KUKA KRL program: MyProgram_222().src

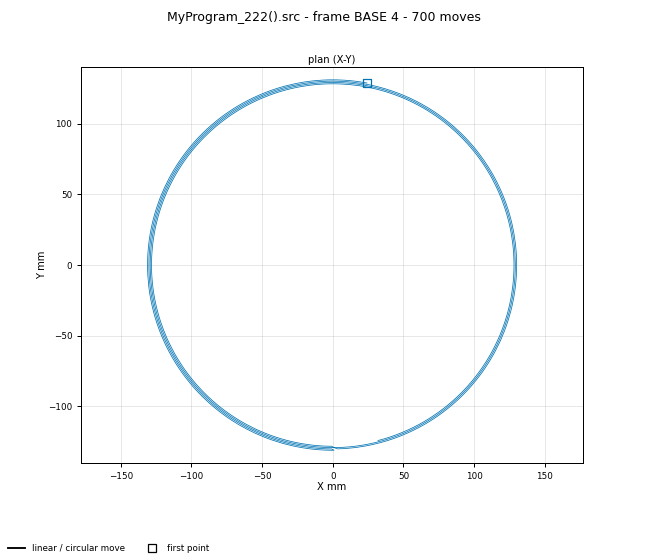
[picture p0: tool path of MyProgram_222().src in frame BASE 4, 700 of 700 moves have a stored position in this frame; points joined in program order, loops and branches not executed]
&ACCESS RVP
&REL 1
&PARAM TEMPLATE = C:\KRC\Roboter\Template\vorgabe
&PARAM EDITMASK = *
DEF MyProgram_222()
; ---- Setting reference (Base) ----
$BASE = BASE_DATA[4]

; --------------------------
; ---- Setting tool (TCP) ----
$TOOL = TOOL_DATA[3]
; --------------------------

$VEL.CP = VEL_APROX_PRINT
Startdeposition()
$VEL.CP = VEL_PRINT
LIN {X 24.2345,Y 128.7731,Z 154,A 76.9385,B 20.8095,C -0.9672,E1 20.8599,E2 370.7346} C_DIS
LIN {X 21.4392,Y 129.2675,Z 154,A 78.2158,B 20.8094,C -0.9692,E1 20.8564,E2 369.4533} C_DIS
LIN {X 16.024,Y 130.0508,Z 154,A 80.7871,B 20.809,C -0.9774,E1 20.8492,E2 366.8615} C_DIS
LIN {X 11.868,Y 130.4964,Z 154,A 82.5489,B 20.8091,C -0.9749,E1 20.8444,E2 365.1082} C_DIS
LIN {X 8.0216,Y 130.7876,Z 154,A 84.1635,B 20.8092,C -0.972,E1 20.8399,E2 363.5027} C_DIS
LIN {X 2.5644,Y 131.0089,Z 154,A 86.3389,B 20.8096,C -0.9629,E1 20.8339,E2 361.3536} C_DIS
LIN {X -2.8562,Y 131.0038,Z 154,A 88.8377,B 20.8094,C -0.9678,E1 20.8269,E2 358.8408} C_DIS
LIN {X -6.3957,Y 130.8773,Z 154,A 90.456,B 20.8094,C -0.9703,E1 20.8224,E2 357.2152} C_DIS
LIN {X -11.494,Y 130.529,Z 154,A 92.9422,B 20.8089,C -0.98,E1 20.8154,E2 354.7005} C_DIS
LIN {X -16.5105,Y 129.9899,Z 154,A 94.7586,B 20.8097,C -0.9625,E1 20.8104,E2 352.9318} C_DIS
LIN {X -20.6648,Y 129.3949,Z 154,A 97.517,B 20.808,C -0.9999,E1 20.8026,E2 350.065} C_DIS
LIN {X -26.2487,Y 128.3772,Z 154,A 99.0193,B 20.8099,C -0.9572,E1 20.7988,E2 348.6809} C_DIS
LIN {X -33.4387,Y 126.695,Z 154,A 102.2474,B 20.81,C -0.9543,E1 20.79,E2 345.456} C_DIS
LIN {X -36.504,Y 125.846,Z 154,A 104.0123,B 20.8094,C -0.9682,E1 20.7851,E2 343.6482} C_DIS
LIN {X -40.1032,Y 124.7455,Z 154,A 105.4729,B 20.8098,C -0.9588,E1 20.7813,E2 342.211} C_DIS
LIN {X -43.2905,Y 123.6759,Z 154,A 106.9808,B 20.8098,C -0.9586,E1 20.7773,E2 340.7001} C_DIS
LIN {X -47.1813,Y 122.2442,Z 154,A 109.222,B 20.8092,C -0.9739,E1 20.7713,E2 338.4101} C_DIS
LIN {X -50.8203,Y 120.7768,Z 154,A 110.8891,B 20.8093,C -0.9696,E1 20.7671,E2 336.7505} C_DIS
LIN {X -54.2769,Y 119.2655,Z 154,A 112.1414,B 20.8102,C -0.9509,E1 20.764,E2 335.5471} C_DIS
LIN {X -56.8312,Y 118.0677,Z 154,A 113.3991,B 20.8102,C -0.9501,E1 20.7608,E2 334.2878} C_DIS
LIN {X -60.4344,Y 116.2651,Z 154,A 115.2346,B 20.8102,C -0.9503,E1 20.7562,E2 332.4457} C_DIS
LIN {X -64.1629,Y 114.2508,Z 154,A 117.1236,B 20.8102,C -0.9487,E1 20.7516,E2 330.5547} C_DIS
LIN {X -68.0819,Y 111.9602,Z 154,A 119.1336,B 20.8104,C -0.9462,E1 20.7468,E2 328.5442} C_DIS
LIN {X -72.0349,Y 109.4582,Z 154,A 120.9854,B 20.8109,C -0.9346,E1 20.7425,E2 326.7178} C_DIS
LIN {X -75.0206,Y 107.4341,Z 154,A 122.714,B 20.8107,C -0.9377,E1 20.7385,E2 324.9735} C_DIS
LIN {X -78.5517,Y 104.8803,Z 154,A 124.7052,B 20.8107,C -0.9373,E1 20.734,E2 322.9747} C_DIS
LIN {X -82.0424,Y 102.1726,Z 154,A 126.6465,B 20.8109,C -0.9336,E1 20.7297,E2 321.0349} C_DIS
LIN {X -85.6297,Y 99.1851,Z 154,A 128.659,B 20.8112,C -0.9281,E1 20.7255,E2 319.0287} C_DIS
LIN {X -88.9399,Y 96.2286,Z 154,A 130.6277,B 20.8112,C -0.9248,E1 20.7214,E2 317.0595} C_DIS
LIN {X -92.1005,Y 93.208,Z 154,A 132.5788,B 20.8114,C -0.9219,E1 20.7175,E2 315.1065} C_DIS
LIN {X -95.171,Y 90.0702,Z 154,A 134.4907,B 20.8116,C -0.917,E1 20.7138,E2 313.1983} C_DIS
LIN {X -98.1976,Y 86.7603,Z 154,A 136.4437,B 20.8118,C -0.9119,E1 20.7102,E2 311.2492} C_DIS
LIN {X -101.0948,Y 83.3668,Z 154,A 138.3845,B 20.8121,C -0.9066,E1 20.7067,E2 309.3126} C_DIS
LIN {X -103.7529,Y 80.0346,Z 154,A 140.297,B 20.8121,C -0.9037,E1 20.7034,E2 307.3972} C_DIS
LIN {X -106.3782,Y 76.511,Z 154,A 142.2645,B 20.8123,C -0.9004,E1 20.7001,E2 305.4272} C_DIS
LIN {X -109.0084,Y 72.7137,Z 154,A 144.2582,B 20.8126,C -0.8939,E1 20.697,E2 303.4398} C_DIS
LIN {X -112.0617,Y 67.9139,Z 154,A 146.7553,B 20.8129,C -0.8874,E1 20.6933,E2 300.9456} C_DIS
LIN {X -114.333,Y 64.0166,Z 154,A 148.7191,B 20.8131,C -0.8814,E1 20.6906,E2 298.986} C_DIS
LIN {X -116.0906,Y 60.7667,Z 154,A 150.2856,B 20.8134,C -0.8749,E1 20.6886,E2 297.4278} C_DIS
LIN {X -119.068,Y 54.704,Z 154,A 153.2497,B 20.8137,C -0.8667,E1 20.685,E2 294.4674} C_DIS
LIN {X -120.3657,Y 51.7859,Z 154,A 154.6481,B 20.8138,C -0.8626,E1 20.6834,E2 293.071} C_DIS
LIN {X -121.5825,Y 48.8605,Z 154,A 156.0604,B 20.814,C -0.8595,E1 20.6819,E2 291.6579} C_DIS
LIN {X -122.8095,Y 45.6896,Z 154,A 157.5478,B 20.8141,C -0.855,E1 20.6805,E2 290.1728} C_DIS
LIN {X -123.9154,Y 42.5996,Z 154,A 158.9849,B 20.8143,C -0.8507,E1 20.6791,E2 288.7378} C_DIS
LIN {X -124.8409,Y 39.8046,Z 154,A 160.2914,B 20.8144,C -0.8476,E1 20.678,E2 287.4313} C_DIS
LIN {X -126.0208,Y 35.9,Z 154,A 162.1837,B 20.8144,C -0.8463,E1 20.6765,E2 285.5291} C_DIS
LIN {X -126.991,Y 32.2948,Z 154,A 163.7475,B 20.8148,C -0.8386,E1 20.6754,E2 283.976} C_DIS
LIN {X -127.8138,Y 28.8687,Z 154,A 165.2513,B 20.815,C -0.8323,E1 20.6745,E2 282.4792} C_DIS
LIN {X -128.4683,Y 25.8008,Z 154,A 166.7991,B 20.815,C -0.8349,E1 20.6736,E2 280.9128} C_DIS
LIN {X -129.3205,Y 21.1211,Z 154,A 168.7012,B 20.8154,C -0.8214,E1 20.6727,E2 279.0351} C_DIS
LIN {X -129.8102,Y 17.8738,Z 154,A 170.3617,B 20.8153,C -0.8256,E1 20.672,E2 277.3505} C_DIS
LIN {X -130.504,Y 11.7863,Z 154,A 173.7319,B 20.8146,C -0.8443,E1 20.6711,E2 273.9024} C_DIS
LIN {X -130.8954,Y 6.0353,Z 154,A 176.4571,B 20.8146,C -0.8445,E1 20.6707,E2 271.1565} C_DIS
LIN {X -131.0326,Y -0.6933,Z 154,A 178.1744,B 20.8167,C -0.7869,E1 20.6707,E2 269.5898} C_DIS
LIN {X -130.843,Y -7.0789,Z 154,A -179.0781,B 20.8171,C -0.7762,E1 20.671,E2 266.8524} C_DIS
LIN {X -130.1846,Y -14.9013,Z 154,A -174.7836,B 20.8163,C -0.7992,E1 20.6721,E2 262.4611} C_DIS
LIN {X -129.629,Y -19.1413,Z 154,A -173.4391,B 20.8172,C -0.7727,E1 20.6726,E2 261.1819} C_DIS
LIN {X -129.0533,Y -22.6958,Z 154,A -171.7247,B 20.8172,C -0.7733,E1 20.6734,E2 259.4532} C_DIS
LIN {X -128.2919,Y -26.6678,Z 154,A -169.9093,B 20.8173,C -0.7697,E1 20.6744,E2 257.6348} C_DIS
LIN {X -127.3798,Y -30.7254,Z 154,A -168.1882,B 20.8177,C -0.7604,E1 20.6755,E2 255.9279} C_DIS
LIN {X -126.5742,Y -33.8918,Z 154,A -166.759,B 20.8178,C -0.7561,E1 20.6765,E2 254.5006} C_DIS
LIN {X -125.6202,Y -37.2753,Z 154,A -165.0809,B 20.8178,C -0.757,E1 20.6778,E2 252.808} C_DIS
LIN {X -124.3719,Y -41.2468,Z 154,A -162.6423,B 20.8171,C -0.7762,E1 20.68,E2 250.2977} C_DIS
LIN {X -122.5336,Y -46.4263,Z 154,A -160.6863,B 20.818,C -0.7514,E1 20.6819,E2 248.3986} C_DIS
LIN {X -120.7003,Y -51.0034,Z 154,A -158.6215,B 20.8183,C -0.7416,E1 20.6841,E2 246.3475} C_DIS
LIN {X -118.8743,Y -55.123,Z 154,A -156.7918,B 20.8187,C -0.7305,E1 20.6861,E2 244.5369} C_DIS
LIN {X -117.4076,Y -58.1818,Z 154,A -155.3038,B 20.8188,C -0.7266,E1 20.688,E2 243.0501} C_DIS
LIN {X -115.5514,Y -61.7905,Z 154,A -152.8099,B 20.818,C -0.7505,E1 20.6914,E2 240.4721} C_DIS
LIN {X -112.948,Y -66.4295,Z 154,A -151.1477,B 20.8191,C -0.7177,E1 20.6936,E2 238.8922} C_DIS
LIN {X -110.8233,Y -69.9165,Z 154,A -149.0444,B 20.8188,C -0.7258,E1 20.6967,E2 236.7529} C_DIS
LIN {X -108.9552,Y -72.7934,Z 154,A -147.8001,B 20.8193,C -0.7118,E1 20.6986,E2 235.5407} C_DIS
LIN {X -106.5761,Y -76.2342,Z 154,A -145.9473,B 20.8194,C -0.7082,E1 20.7016,E2 233.6869} C_DIS
LIN {X -103.944,Y -79.7861,Z 154,A -144.0006,B 20.8195,C -0.7041,E1 20.7049,E2 231.7405} C_DIS
LIN {X -100.9127,Y -83.5867,Z 154,A -142.0048,B 20.8199,C -0.6938,E1 20.7083,E2 229.7622} C_DIS
LIN {X -98.5369,Y -86.3752,Z 154,A -140.2377,B 20.8198,C -0.6969,E1 20.7116,E2 227.9767} C_DIS
LIN {X -95.6003,Y -89.6151,Z 154,A -138.2924,B 20.8198,C -0.694,E1 20.7153,E2 226.029} C_DIS
LIN {X -92.5258,Y -92.7855,Z 154,A -136.3824,B 20.82,C -0.6891,E1 20.719,E2 224.123} C_DIS
LIN {X -87.9892,Y -97.098,Z 154,A -133.6886,B 20.8203,C -0.6817,E1 20.7245,E2 221.4364} C_DIS
LIN {X -84.929,Y -99.7857,Z 154,A -131.8372,B 20.8203,C -0.6812,E1 20.7284,E2 219.5777} C_DIS
LIN {X -81.3185,Y -102.7499,Z 154,A -129.9267,B 20.8206,C -0.672,E1 20.7325,E2 217.6844} C_DIS
LIN {X -78.4497,Y -104.9562,Z 154,A -128.241,B 20.8206,C -0.6735,E1 20.7363,E2 215.9871} C_DIS
LIN {X -74.5643,Y -107.7516,Z 154,A -126.134,B 20.8206,C -0.6705,E1 20.7411,E2 213.8795} C_DIS
LIN {X -71.0131,Y -110.1245,Z 154,A -123.6707,B 20.8199,C -0.6923,E1 20.7471,E2 211.3449} C_DIS
LIN {X -66.7684,Y -112.7486,Z 154,A -122.2996,B 20.8211,C -0.6554,E1 20.7501,E2 210.0728} C_DIS
LIN {X -64.3749,Y -114.1316,Z 154,A -120.804,B 20.8208,C -0.6656,E1 20.7538,E2 208.5431} C_DIS
LIN {X -60.4908,Y -116.2355,Z 154,A -118.9918,B 20.821,C -0.6581,E1 20.7582,E2 206.7458} C_DIS
LIN {X -57.2733,Y -117.8555,Z 154,A -117.4224,B 20.821,C -0.6559,E1 20.7622,E2 205.1776} C_DIS
LIN {X -54.7452,Y -119.0489,Z 154,A -116.1375,B 20.821,C -0.6571,E1 20.7654,E2 203.8853} C_DIS
LIN {X -48.5369,Y -121.7129,Z 154,A -113.2537,B 20.8212,C -0.6511,E1 20.7729,E2 201.0106} C_DIS
LIN {X -45.8983,Y -122.7313,Z 154,A -111.9528,B 20.8212,C -0.6526,E1 20.7763,E2 199.7019} C_DIS
LIN {X -42.6798,Y -123.8876,Z 154,A -110.4471,B 20.8212,C -0.6517,E1 20.7802,E2 198.1951} C_DIS
LIN {X -38.7276,Y -125.1798,Z 154,A -108.5832,B 20.8212,C -0.6523,E1 20.7852,E2 196.3257} C_DIS
LIN {X -35.9482,Y -126.0073,Z 154,A -107.2661,B 20.8212,C -0.6534,E1 20.7888,E2 195.0027} C_DIS
LIN {X -31.8644,Y -127.1002,Z 154,A -105.6338,B 20.8214,C -0.6432,E1 20.7931,E2 193.3963} C_DIS
LIN {X -29.3432,Y -127.7054,Z 154,A -104.4238,B 20.8214,C -0.6458,E1 20.7964,E2 192.1769} C_DIS
LIN {X -26.05,Y -128.4176,Z 154,A -102.9176,B 20.8214,C -0.6465,E1 20.8005,E2 190.6665} C_DIS
LIN {X -22.3946,Y -129.1072,Z 154,A -100.5403,B 20.8204,C -0.6781,E1 20.8073,E2 188.1974} C_DIS
LIN {X -17.021,Y -129.923,Z 154,A -99.0918,B 20.8216,C -0.6377,E1 20.811,E2 186.8613} C_DIS
LIN {X -13.986,Y -130.2847,Z 154,A -97.5622,B 20.8214,C -0.6457,E1 20.8153,E2 185.3079} C_DIS
LIN {X -9.9937,Y -130.6525,Z 154,A -95.756,B 20.8213,C -0.6479,E1 20.8204,E2 183.4946} C_DIS
LIN {X -6.1332,Y -130.8905,Z 154,A -94.0071,B 20.8213,C -0.6504,E1 20.8253,E2 181.7381} C_DIS
LIN {X -2.0568,Y -131.0173,Z 154,A -92.3251,B 20.8213,C -0.6463,E1 20.8299,E2 180.0675} C_DIS
LIN {X 0.9184,Y -131.027,Z 154,A -91.2855,B 20.8217,C -0.6353,E1 20.8328,E2 179.0588} C_DIS
Enddeposition()
LIN {X 0.9184,Y -131.027,Z 154,A -91.2855,B 20.8217,C -0.6353,E1 20.8328,E2 179.0588} C_DIS
Startdeposition()
$VEL.CP = VEL_PRINT
LIN {X -0.7968,Y -130.0933,Z 154,A -92.0736,B 19.5759,C -0.4592,E1 19.5796,E2 180.2341} C_DIS
LIN {X -4.6188,Y -130.0145,Z 154,A -93.836,B 19.576,C -0.4559,E1 19.5747,E2 182.0066} C_DIS
LIN {X -8.3305,Y -129.8291,Z 154,A -95.4802,B 19.576,C -0.4556,E1 19.5701,E2 183.6523} C_DIS
LIN {X -12.3798,Y -129.5053,Z 154,A -97.2178,B 19.576,C -0.4578,E1 19.5653,E2 185.3845} C_DIS
LIN {X -15.9258,Y -129.1181,Z 154,A -98.8616,B 19.576,C -0.4552,E1 19.5607,E2 187.0374} C_DIS
LIN {X -22.7172,Y -128.0969,Z 154,A -101.5472,B 19.5757,C -0.4694,E1 19.5534,E2 189.6837} C_DIS
LIN {X -27.1192,Y -127.2379,Z 154,A -103.7303,B 19.5759,C -0.4621,E1 19.5473,E2 191.8919} C_DIS
LIN {X -30.0781,Y -126.5713,Z 154,A -105.1453,B 19.5759,C -0.4597,E1 19.5435,E2 193.3164} C_DIS
LIN {X -33.666,Y -125.6639,Z 154,A -106.7262,B 19.5759,C -0.4626,E1 19.5392,E2 194.8917} C_DIS
LIN {X -37.1625,Y -124.6762,Z 154,A -108.5748,B 19.5761,C -0.4541,E1 19.5342,E2 196.7697} C_DIS
LIN {X -41.5663,Y -123.2772,Z 154,A -110.3638,B 19.5758,C -0.4652,E1 19.5295,E2 198.5297} C_DIS
LIN {X -44.5248,Y -122.2395,Z 154,A -111.7569,B 19.5758,C -0.4659,E1 19.5258,E2 199.9242} C_DIS
LIN {X -48.0211,Y -120.9098,Z 154,A -113.5186,B 19.5758,C -0.4631,E1 19.5212,E2 201.6992} C_DIS
LIN {X -53.3422,Y -118.6568,Z 154,A -115.9843,B 19.5758,C -0.4689,E1 19.5149,E2 204.1552} C_DIS
LIN {X -57.333,Y -116.7807,Z 154,A -117.6902,B 19.5755,C -0.4802,E1 19.5107,E2 205.8329} C_DIS
LIN {X -59.8031,Y -115.5375,Z 154,A -119.207,B 19.5757,C -0.4703,E1 19.5068,E2 207.3848} C_DIS
LIN {X -63.2265,Y -113.7001,Z 154,A -120.9707,B 19.5757,C -0.4706,E1 19.5025,E2 209.1541} C_DIS
LIN {X -69.7369,Y -109.8275,Z 154,A -124.276,B 19.5755,C -0.4766,E1 19.4946,E2 212.4546} C_DIS
LIN {X -72.7821,Y -107.8334,Z 154,A -126.1024,B 19.5757,C -0.4708,E1 19.4903,E2 214.3065} C_DIS
LIN {X -75.9627,Y -105.6175,Z 154,A -127.6621,B 19.5755,C -0.4791,E1 19.4868,E2 215.8483} C_DIS
LIN {X -79.3729,Y -103.0794,Z 154,A -129.5394,B 19.5755,C -0.4822,E1 19.4826,E2 217.7252} C_DIS
LIN {X -82.4141,Y -100.6637,Z 154,A -131.0389,B 19.5752,C -0.4932,E1 19.4794,E2 219.199} C_DIS
LIN {X -85.1425,Y -98.3673,Z 154,A -132.8193,B 19.5752,C -0.4884,E1 19.4756,E2 221.003} C_DIS
LIN {X -88.6083,Y -95.2564,Z 154,A -135.2225,B 19.5755,C -0.4794,E1 19.4706,E2 223.4459} C_DIS
LIN {X -91.4633,Y -92.5194,Z 154,A -136.6252,B 19.5751,C -0.4955,E1 19.4678,E2 224.808} C_DIS
LIN {X -94.3948,Y -89.5265,Z 154,A -138.5245,B 19.5751,C -0.4974,E1 19.4642,E2 226.7122} C_DIS
LIN {X -96.7023,Y -87.0288,Z 154,A -140.0164,B 19.575,C -0.5009,E1 19.4614,E2 228.2023} C_DIS
LIN {X -99.6079,Y -83.6871,Z 154,A -141.9787,B 19.5749,C -0.5049,E1 19.4578,E2 230.1644} C_DIS
LIN {X -102.3115,Y -80.3593,Z 154,A -143.5791,B 19.5745,C -0.5199,E1 19.4551,E2 231.7295} C_DIS
LIN {X -104.2104,Y -77.8814,Z 154,A -145.1638,B 19.5746,C -0.5154,E1 19.4523,E2 233.3376} C_DIS
LIN {X -106.4422,Y -74.8022,Z 154,A -146.913,B 19.5746,C -0.5168,E1 19.4495,E2 235.0939} C_DIS
LIN {X -109.4461,Y -70.3339,Z 154,A -149.0586,B 19.5742,C -0.531,E1 19.4462,E2 237.2108} C_DIS
LIN {X -111.1086,Y -67.6779,Z 154,A -150.735,B 19.5744,C -0.5237,E1 19.4437,E2 238.9203} C_DIS
LIN {X -114.5747,Y -61.6271,Z 154,A -153.7303,B 19.5741,C -0.5346,E1 19.4396,E2 241.9036} C_DIS
LIN {X -116.1029,Y -58.6942,Z 154,A -155.149,B 19.574,C -0.5399,E1 19.4378,E2 243.3163} C_DIS
LIN {X -117.7336,Y -55.3547,Z 154,A -157.0339,B 19.574,C -0.5354,E1 19.4355,E2 245.2281} C_DIS
LIN {X -119.3563,Y -51.7577,Z 154,A -158.5683,B 19.5738,C -0.5477,E1 19.4338,E2 246.7368} C_DIS
LIN {X -120.7066,Y -48.5252,Z 154,A -160.1708,B 19.5738,C -0.5499,E1 19.4321,E2 248.3444} C_DIS
LIN {X -122.6109,Y -43.4932,Z 154,A -162.7628,B 19.5738,C -0.5487,E1 19.4296,E2 250.9592} C_DIS
LIN {X -123.9948,Y -39.3717,Z 154,A -164.4736,B 19.5734,C -0.5616,E1 19.4281,E2 252.644} C_DIS
LIN {X -125.2191,Y -35.2852,Z 154,A -166.3449,B 19.5732,C -0.5674,E1 19.4267,E2 254.512} C_DIS
LIN {X -126.1307,Y -31.8726,Z 154,A -167.8804,B 19.5731,C -0.5728,E1 19.4256,E2 256.0431} C_DIS
LIN {X -126.911,Y -28.6103,Z 154,A -169.3933,B 19.573,C -0.576,E1 19.4246,E2 257.5582} C_DIS
LIN {X -127.7734,Y -24.4702,Z 154,A -171.2768,B 19.5728,C -0.5809,E1 19.4236,E2 259.4415} C_DIS
LIN {X -128.4637,Y -20.5514,Z 154,A -173.1459,B 19.5728,C -0.582,E1 19.4227,E2 261.3217} C_DIS
LIN {X -129.1831,Y -15.3814,Z 154,A -175.7232,B 19.5728,C -0.5792,E1 19.4218,E2 263.9277} C_DIS
LIN {X -129.5709,Y -11.6949,Z 154,A -177.088,B 19.5725,C -0.5938,E1 19.4215,E2 265.2595} C_DIS
LIN {X -129.8563,Y -7.8883,Z 154,A -178.7027,B 19.5722,C -0.6014,E1 19.4212,E2 266.864} C_DIS
LIN {X -130.084,Y -1.7845,Z 154,A 178.548,B 19.5721,C -0.6077,E1 19.4209,E2 269.6162} C_DIS
LIN {X -129.9989,Y 5.017,Z 154,A 175.5447,B 19.5718,C -0.6168,E1 19.4211,E2 272.6159} C_DIS
LIN {X -129.6293,Y 11.0053,Z 154,A 172.7722,B 19.5717,C -0.6204,E1 19.4216,E2 275.3993} C_DIS
LIN {X -129.2066,Y 15.1843,Z 154,A 171.0134,B 19.5714,C -0.6294,E1 19.4221,E2 277.1448} C_DIS
LIN {X -128.7288,Y 18.8128,Z 154,A 169.4742,B 19.5712,C -0.637,E1 19.4227,E2 278.6732} C_DIS
LIN {X -128.2265,Y 21.9802,Z 154,A 167.7311,B 19.5714,C -0.6297,E1 19.4235,E2 280.4521} C_DIS
LIN {X -127.4357,Y 26.1728,Z 154,A 166.0763,B 19.571,C -0.6435,E1 19.4244,E2 282.0782} C_DIS
LIN {X -126.5199,Y 30.2914,Z 154,A 164.1884,B 19.5708,C -0.6481,E1 19.4256,E2 283.9666} C_DIS
LIN {X -125.6596,Y 33.6822,Z 154,A 162.6937,B 19.5706,C -0.6545,E1 19.4267,E2 285.4536} C_DIS
LIN {X -124.6598,Y 37.2182,Z 154,A 160.8958,B 19.5706,C -0.653,E1 19.4281,E2 287.2696} C_DIS
LIN {X -123.5026,Y 40.8893,Z 154,A 159.3203,B 19.5704,C -0.6624,E1 19.4294,E2 288.8286} C_DIS
LIN {X -122.3999,Y 44.08,Z 154,A 157.8409,B 19.5702,C -0.6672,E1 19.4308,E2 290.3048} C_DIS
LIN {X -121.2033,Y 47.2711,Z 154,A 156.3548,B 19.57,C -0.6721,E1 19.4323,E2 291.7869} C_DIS
LIN {X -119.8982,Y 50.4909,Z 154,A 154.804,B 19.57,C -0.6759,E1 19.4339,E2 293.3377} C_DIS
LIN {X -118.5097,Y 53.6711,Z 154,A 153.1694,B 19.5699,C -0.6766,E1 19.4358,E2 294.9822} C_DIS
LIN {X -116.548,Y 57.8048,Z 154,A 151.2069,B 19.5696,C -0.6843,E1 19.4381,E2 296.9354} C_DIS
LIN {X -114.1362,Y 62.4356,Z 154,A 149.0496,B 19.5692,C -0.6959,E1 19.4409,E2 299.0729} C_DIS
LIN {X -112.6163,Y 65.137,Z 154,A 147.2617,B 19.5696,C -0.6845,E1 19.4435,E2 300.9072} C_DIS
LIN {X -109.7751,Y 69.8199,Z 154,A 145.1433,B 19.569,C -0.7017,E1 19.4465,E2 302.9883} C_DIS
LIN {X -107.9103,Y 72.6686,Z 154,A 143.4595,B 19.5691,C -0.6991,E1 19.4492,E2 304.6909} C_DIS
LIN {X -105.3906,Y 76.2764,Z 154,A 141.5211,B 19.569,C -0.7042,E1 19.4523,E2 306.6264} C_DIS
LIN {X -102.7987,Y 79.7351,Z 154,A 139.6252,B 19.5688,C -0.7094,E1 19.4555,E2 308.5186} C_DIS
LIN {X -100.0247,Y 83.1888,Z 154,A 137.6414,B 19.5686,C -0.7131,E1 19.459,E2 310.5034} C_DIS
LIN {X -97.1668,Y 86.5102,Z 154,A 135.6917,B 19.5686,C -0.7171,E1 19.4626,E2 312.4526} C_DIS
LIN {X -94.2861,Y 89.6409,Z 154,A 133.7809,B 19.5684,C -0.7202,E1 19.4662,E2 314.3649} C_DIS
LIN {X -91.1498,Y 92.8277,Z 154,A 131.835,B 19.5682,C -0.7256,E1 19.4701,E2 316.3053} C_DIS
LIN {X -87.8572,Y 95.9501,Z 154,A 129.8474,B 19.568,C -0.7305,E1 19.4741,E2 318.289} C_DIS
LIN {X -84.5917,Y 98.8416,Z 154,A 127.8591,B 19.568,C -0.7322,E1 19.4783,E2 320.2825} C_DIS
LIN {X -81.2047,Y 101.6421,Z 154,A 125.9265,B 19.5678,C -0.7363,E1 19.4825,E2 322.2122} C_DIS
LIN {X -77.6411,Y 104.3893,Z 154,A 123.9747,B 19.5676,C -0.7414,E1 19.4868,E2 324.158} C_DIS
LIN {X -74.0496,Y 106.9673,Z 154,A 122.0132,B 19.5676,C -0.7446,E1 19.4913,E2 326.1186} C_DIS
LIN {X -70.5255,Y 109.3231,Z 154,A 120.1466,B 19.5674,C -0.7481,E1 19.4956,E2 327.9829} C_DIS
LIN {X -67.5488,Y 111.1868,Z 154,A 118.5412,B 19.5674,C -0.7486,E1 19.4995,E2 329.5932} C_DIS
LIN {X -63.5466,Y 113.5215,Z 154,A 116.4535,B 19.5674,C -0.7503,E1 19.5045,E2 331.6839} C_DIS
LIN {X -60.1354,Y 115.363,Z 154,A 114.917,B 19.567,C -0.7594,E1 19.5083,E2 333.1989} C_DIS
LIN {X -57.3969,Y 116.7492,Z 154,A 113.5105,B 19.567,C -0.7594,E1 19.5118,E2 334.6101} C_DIS
LIN {X -54.2142,Y 118.2614,Z 154,A 111.873,B 19.567,C -0.7585,E1 19.516,E2 336.2558} C_DIS
LIN {X -47.52,Y 121.1065,Z 154,A 108.937,B 19.5665,C -0.7727,E1 19.5234,E2 339.1578} C_DIS
LIN {X -43.9789,Y 122.4364,Z 154,A 107.1001,B 19.5666,C -0.7683,E1 19.5283,E2 341.0128} C_DIS
LIN {X -40.4453,Y 123.6505,Z 154,A 105.2969,B 19.5668,C -0.7643,E1 19.5331,E2 342.8326} C_DIS
LIN {X -36.3926,Y 124.9016,Z 154,A 103.5536,B 19.5665,C -0.7709,E1 19.5377,E2 344.5598} C_DIS
LIN {X -33.0324,Y 125.8329,Z 154,A 101.4958,B 19.5672,C -0.7527,E1 19.5435,E2 346.6761} C_DIS
LIN {X -28.8174,Y 126.8637,Z 154,A 100.1247,B 19.5664,C -0.7747,E1 19.547,E2 347.9839} C_DIS
LIN {X -20.5245,Y 128.4678,Z 154,A 96.4736,B 19.5662,C -0.7799,E1 19.557,E2 351.6244} C_DIS
LIN {X -14.0527,Y 129.3345,Z 154,A 93.5362,B 19.5662,C -0.7791,E1 19.5652,E2 354.567} C_DIS
LIN {X -7.971,Y 129.8512,Z 154,A 90.8212,B 19.5662,C -0.7791,E1 19.5727,E2 357.2835} C_DIS
LIN {X -4.3216,Y 130.0254,Z 154,A 88.6931,B 19.567,C -0.7596,E1 19.5788,E2 359.4703} C_DIS
LIN {X -0.0103,Y 130.0977,Z 154,A 87.2915,B 19.5662,C -0.779,E1 19.5826,E2 360.8141} C_DIS
LIN {X 6.3432,Y 129.9411,Z 154,A 84.4877,B 19.5662,C -0.779,E1 19.5904,E2 363.6171} C_DIS
LIN {X 10.1006,Y 129.7045,Z 154,A 82.584,B 19.5666,C -0.7692,E1 19.5958,E2 365.5486} C_DIS
LIN {X 14.7181,Y 129.2622,Z 154,A 80.0681,B 19.5673,C -0.7505,E1 19.6029,E2 368.1179} C_DIS
LIN {X 20.0105,Y 128.5474,Z 154,A 78.5006,B 19.5662,C -0.7803,E1 19.607,E2 369.5947} C_DIS
LIN {X 25.0067,Y 127.6708,Z 154,A 76.1154,B 19.5664,C -0.7734,E1 19.6136,E2 371.997} C_DIS
LIN {X 29.4238,Y 126.7252,Z 154,A 74.2706,B 19.5663,C -0.778,E1 19.6186,E2 373.8247} C_DIS
LIN {X 32.4616,Y 125.9813,Z 154,A 72.7792,B 19.5665,C -0.7726,E1 19.6226,E2 375.3292} C_DIS
LIN {X 37.2829,Y 124.6409,Z 154,A 70.6886,B 19.5664,C -0.7755,E1 19.6282,E2 377.4066} C_DIS
LIN {X 40.1199,Y 123.7558,Z 154,A 69.3852,B 19.5664,C -0.7747,E1 19.6317,E2 378.7093} C_DIS
LIN {X 43.0059,Y 122.7821,Z 154,A 67.8929,B 19.5667,C -0.7675,E1 19.6357,E2 380.2191} C_DIS
LIN {X 46.6129,Y 121.4583,Z 154,A 65.8639,B 19.5672,C -0.7525,E1 19.6411,E2 382.2871} C_DIS
LIN {X 50.3714,Y 119.9481,Z 154,A 64.514,B 19.5667,C -0.7678,E1 19.6444,E2 383.5871} C_DIS
LIN {X 55.0036,Y 117.8964,Z 154,A 62.2453,B 19.5668,C -0.7638,E1 19.6502,E2 385.8605} C_DIS
LIN {X 59.3937,Y 115.7468,Z 154,A 60.2443,B 19.5667,C -0.7671,E1 19.6552,E2 387.8444} C_DIS
LIN {X 62.1329,Y 114.3013,Z 154,A 58.5729,B 19.5672,C -0.7529,E1 19.6594,E2 389.5519} C_DIS
LIN {X 67.9937,Y 110.9149,Z 154,A 56.134,B 19.5666,C -0.7705,E1 19.6651,E2 391.9287} C_DIS
LIN {X 72.3556,Y 108.1201,Z 154,A 53.5799,B 19.5671,C -0.7558,E1 19.6712,E2 394.5156} C_DIS
LIN {X 75.5322,Y 105.9253,Z 154,A 51.8025,B 19.5673,C -0.7498,E1 19.6752,E2 396.3028} C_DIS
LIN {X 79.0736,Y 103.3084,Z 154,A 49.8749,B 19.5674,C -0.7469,E1 19.6795,E2 398.2299} C_DIS
LIN {X 82.6183,Y 100.4969,Z 154,A 47.8799,B 19.5676,C -0.7431,E1 19.6839,E2 400.2264} C_DIS
LIN {X 85.8532,Y 97.7478,Z 154,A 45.9939,B 19.5677,C -0.7388,E1 19.6879,E2 402.1154} C_DIS
LIN {X 90.4931,Y 93.4679,Z 154,A 43.2586,B 19.5679,C -0.735,E1 19.6934,E2 404.8473} C_DIS
LIN {X 93.5957,Y 90.3611,Z 154,A 41.3568,B 19.5679,C -0.7322,E1 19.6972,E2 406.7468} C_DIS
LIN {X 96.4516,Y 87.3062,Z 154,A 39.5084,B 19.5681,C -0.7278,E1 19.7007,E2 408.5974} C_DIS
LIN {X 99.2854,Y 84.0698,Z 154,A 37.3833,B 19.5686,C -0.714,E1 19.7046,E2 410.7509} C_DIS
LIN {X 101.4305,Y 81.4689,Z 154,A 36.2251,B 19.5683,C -0.724,E1 19.7065,E2 411.8723} C_DIS
LIN {X 103.8606,Y 78.3469,Z 154,A 34.4104,B 19.5685,C -0.7169,E1 19.7096,E2 413.697} C_DIS
LIN {X 106.964,Y 74.053,Z 154,A 31.8563,B 19.569,C -0.7019,E1 19.7138,E2 416.2791} C_DIS
LIN {X 108.8961,Y 71.1833,Z 154,A 30.8452,B 19.5684,C -0.7194,E1 19.7153,E2 417.2316} C_DIS
LIN {X 110.4165,Y 68.8002,Z 154,A 29.3247,B 19.5689,C -0.7047,E1 19.7176,E2 418.7857} C_DIS
LIN {X 112.3531,Y 65.5909,Z 154,A 27.7185,B 19.569,C -0.7023,E1 19.7199,E2 420.3885} C_DIS
LIN {X 114.4272,Y 61.9017,Z 154,A 25.8198,B 19.5692,C -0.6958,E1 19.7224,E2 422.2932} C_DIS
LIN {X 116.3163,Y 58.2744,Z 154,A 23.5423,B 19.5701,C -0.671,E1 19.7254,E2 424.6284} C_DIS
LIN {X 118.3968,Y 53.9213,Z 154,A 21.945,B 19.5695,C -0.6872,E1 19.7272,E2 426.1665} C_DIS
LIN {X 120.1467,Y 49.896,Z 154,A 20.22,B 19.5695,C -0.6905,E1 19.729,E2 427.8691} C_DIS
LIN {X 121.3083,Y 47.0009,Z 154,A 18.7898,B 19.5696,C -0.6842,E1 19.7305,E2 429.3077} C_DIS
LIN {X 122.4691,Y 43.8879,Z 154,A 17.3036,B 19.5698,C -0.679,E1 19.7319,E2 430.7985} C_DIS
LIN {X 123.7841,Y 40.0312,Z 154,A 15.4757,B 19.57,C -0.6724,E1 19.7336,E2 432.6325} C_DIS
LIN {X 124.854,Y 36.5552,Z 154,A 13.9249,B 19.5701,C -0.6698,E1 19.7348,E2 434.1794} C_DIS
LIN {X 125.8628,Y 32.9202,Z 154,A 11.8618,B 19.5708,C -0.6478,E1 19.7363,E2 436.2919} C_DIS
LIN {X 126.7769,Y 29.1974,Z 154,A 10.6024,B 19.5704,C -0.6609,E1 19.7371,E2 437.5032} C_DIS
LIN {X 128.0681,Y 22.8777,Z 154,A 7.8687,B 19.5705,C -0.6568,E1 19.7386,E2 440.2282} C_DIS
LIN {X 129.2393,Y 14.9106,Z 154,A 3.7241,B 19.5717,C -0.6205,E1 19.7402,E2 444.4483} C_DIS
LIN {X 129.6858,Y 10.3362,Z 154,A 2.3372,B 19.571,C -0.6412,E1 19.7405,E2 445.7631} C_DIS
LIN {X 129.8981,Y 7.1966,Z 154,A 0.3194,B 19.572,C -0.61,E1 19.7408,E2 447.8574} C_DIS
LIN {X 130.071,Y 2.5695,Z 154,A -0.9998,B 19.5713,C -0.6342,E1 19.7409,E2 449.0948} C_DIS
LIN {X 130.0972,Y -0.3469,Z 154,A -2.4781,B 19.5716,C -0.6219,E1 19.7409,E2 450.598} C_DIS
LIN {X 130.0317,Y -4.1113,Z 154,A -4.1517,B 19.5718,C -0.6161,E1 19.7408,E2 452.2759} C_DIS
LIN {X 129.8367,Y -8.2072,Z 154,A -5.8289,B 19.5718,C -0.6159,E1 19.7405,E2 453.9406} C_DIS
LIN {X 129.45,Y -12.9481,Z 154,A -8.4158,B 19.5726,C -0.5884,E1 19.7399,E2 456.5888} C_DIS
LIN {X 128.9509,Y -17.2229,Z 154,A -9.6494,B 19.572,C -0.6106,E1 19.7395,E2 457.7471} C_DIS
LIN {X 128.221,Y -22.0135,Z 154,A -12.0156,B 19.5725,C -0.594,E1 19.7384,E2 460.1443} C_DIS
LIN {X 127.6992,Y -24.8583,Z 154,A -13.7138,B 19.5731,C -0.572,E1 19.7375,E2 461.8946} C_DIS
LIN {X 126.7691,Y -29.2315,Z 154,A -15.0447,B 19.5725,C -0.5931,E1 19.7367,E2 463.1531} C_DIS
LIN {X 126.0433,Y -32.2171,Z 154,A -16.4871,B 19.5727,C -0.5851,E1 19.7357,E2 464.6083} C_DIS
LIN {X 124.1684,Y -38.828,Z 154,A -19.4363,B 19.5729,C -0.5791,E1 19.7334,E2 467.5532} C_DIS
LIN {X 122.8883,Y -42.6997,Z 154,A -21.2732,B 19.5731,C -0.5719,E1 19.7318,E2 469.3977} C_DIS
LIN {X 121.4731,Y -46.5771,Z 154,A -23.85,B 19.5741,C -0.5344,E1 19.7291,E2 472.067} C_DIS
LIN {X 119.2962,Y -51.8967,Z 154,A -25.5088,B 19.5733,C -0.5638,E1 19.7274,E2 473.6267} C_DIS
LIN {X 118.0667,Y -54.6353,Z 154,A -27.8975,B 19.5746,C -0.5149,E1 19.7245,E2 476.1434} C_DIS
LIN {X 114.9727,Y -60.8787,Z 154,A -29.9479,B 19.5737,C -0.549,E1 19.722,E2 478.0786} C_DIS
LIN {X 112.8579,Y -64.7182,Z 154,A -31.9333,B 19.5739,C -0.5412,E1 19.7192,E2 480.0737} C_DIS
LIN {X 110.6474,Y -68.4291,Z 154,A -33.835,B 19.5741,C -0.5359,E1 19.7165,E2 481.9782} C_DIS
LIN {X 108.3081,Y -72.0739,Z 154,A -35.7116,B 19.5741,C -0.532,E1 19.7136,E2 483.8541} C_DIS
LIN {X 105.7736,Y -75.7444,Z 154,A -38.0252,B 19.5747,C -0.5121,E1 19.7098,E2 486.212} C_DIS
LIN {X 103.3691,Y -78.9942,Z 154,A -39.2728,B 19.5742,C -0.5299,E1 19.7078,E2 487.3991} C_DIS
LIN {X 101.2869,Y -81.6469,Z 154,A -40.9027,B 19.5745,C -0.52,E1 19.7049,E2 489.0485} C_DIS
LIN {X 97.5417,Y -86.0865,Z 154,A -43.5278,B 19.5747,C -0.5107,E1 19.7001,E2 491.6853} C_DIS
LIN {X 94.6829,Y -89.2211,Z 154,A -45.2658,B 19.5747,C -0.5117,E1 19.6969,E2 493.4104} C_DIS
LIN {X 91.7273,Y -92.257,Z 154,A -47.5265,B 19.5752,C -0.4908,E1 19.6923,E2 495.7205} C_DIS
LIN {X 88.7925,Y -95.085,Z 154,A -49.0355,B 19.575,C -0.4986,E1 19.6893,E2 497.1982} C_DIS
LIN {X 84.9896,Y -98.4989,Z 154,A -51.1695,B 19.575,C -0.4986,E1 19.6848,E2 499.3215} C_DIS
LIN {X 81.6838,Y -101.2572,Z 154,A -53.6675,B 19.5757,C -0.4695,E1 19.6793,E2 501.8932} C_DIS
LIN {X 77.512,Y -104.4854,Z 154,A -55.1265,B 19.575,C -0.5006,E1 19.6762,E2 503.2529} C_DIS
LIN {X 74.8281,Y -106.4239,Z 154,A -56.7892,B 19.5752,C -0.4892,E1 19.6724,E2 504.9419} C_DIS
LIN {X 71.4758,Y -108.7036,Z 154,A -58.5589,B 19.5753,C -0.4865,E1 19.6683,E2 506.7119} C_DIS
LIN {X 68.0217,Y -110.8977,Z 154,A -60.3845,B 19.5754,C -0.4822,E1 19.664,E2 508.5424} C_DIS
LIN {X 64.1761,Y -113.1671,Z 154,A -62.3497,B 19.5754,C -0.4789,E1 19.6592,E2 510.5098} C_DIS
LIN {X 60.779,Y -115.0251,Z 154,A -64.4248,B 19.5759,C -0.4609,E1 19.654,E2 512.6306} C_DIS
LIN {X 57.1038,Y -116.8937,Z 154,A -66.1038,B 19.5759,C -0.4637,E1 19.6498,E2 514.2954} C_DIS
LIN {X 53.9076,Y -118.4032,Z 154,A -67.5369,B 19.5758,C -0.4664,E1 19.6462,E2 515.7156} C_DIS
LIN {X 48.4834,Y -120.7235,Z 154,A -69.9124,B 19.5757,C -0.472,E1 19.6401,E2 518.0673} C_DIS
LIN {X 45.4928,Y -121.8819,Z 154,A -71.2918,B 19.5757,C -0.4715,E1 19.6365,E2 519.4443} C_DIS
LIN {X 42.4766,Y -122.9656,Z 154,A -72.7095,B 19.5757,C -0.4696,E1 19.6328,E2 520.864} C_DIS
LIN {X 38.8379,Y -124.1644,Z 154,A -75.1364,B 19.5764,C -0.4377,E1 19.6261,E2 523.3798} C_DIS
LIN {X 33.6692,Y -125.6631,Z 154,A -76.49,B 19.5756,C -0.4764,E1 19.6228,E2 524.6153} C_DIS
LIN {X 27.4504,Y -127.1664,Z 154,A -79.9627,B 19.5762,C -0.4474,E1 19.6131,E2 528.1681} C_DIS
LIN {X 23.7107,Y -127.9186,Z 154,A -82.0924,B 19.5766,C -0.4282,E1 19.6071,E2 530.3519} C_DIS
LIN {X 17.8454,Y -128.867,Z 154,A -83.7997,B 19.5759,C -0.4628,E1 19.6027,E2 531.954} C_DIS
LIN {X 14.9272,Y -129.2373,Z 154,A -85.3186,B 19.5761,C -0.4531,E1 19.5984,E2 533.5003} C_DIS
LIN {X 10.7067,Y -129.6545,Z 154,A -87.0046,B 19.5759,C -0.4595,E1 19.5938,E2 535.1659} C_DIS
LIN {X 7.1387,Y -129.9011,Z 154,A -88.6911,B 19.5761,C -0.4544,E1 19.589,E2 536.8666} C_DIS
LIN {X 3.335,Y -130.0533,Z 154,A -90.3616,B 19.5761,C -0.4542,E1 19.5844,E2 538.5373} C_DIS
LIN {X 3.335,Y -130.0533,Z 154,A -90.3616,B 19.5761,C -0.4542,E1 19.5844,E2 538.5373} C_DIS
Enddeposition()
LIN {X 0.9058,Y -129.1537,Z 154,A -89.8894,B 16.8368,C -0.1758,E1 16.8403,E2 538.7346} C_DIS
Startdeposition()
$VEL.CP = VEL_PRINT
LIN {X 4.808,Y -129.0687,Z 154,A -88.1118,B 16.8368,C -0.1778,E1 16.8453,E2 536.9507} C_DIS
LIN {X 7.7984,Y -128.9224,Z 154,A -86.7926,B 16.8368,C -0.178,E1 16.849,E2 535.6317} C_DIS
LIN {X 11.9397,Y -128.6055,Z 154,A -84.5096,B 16.8367,C -0.1941,E1 16.8555,E2 533.2952} C_DIS
LIN {X 15.7978,Y -128.1891,Z 154,A -83.2594,B 16.8368,C -0.1785,E1 16.8588,E2 532.1001} C_DIS
LIN {X 20.563,Y -127.5119,Z 154,A -80.6264,B 16.8366,C -0.1973,E1 16.8662,E2 529.4063} C_DIS
LIN {X 24.4435,Y -126.8238,Z 154,A -79.3968,B 16.8368,C -0.1804,E1 16.8695,E2 528.2372} C_DIS
LIN {X 30.435,Y -125.5207,Z 154,A -76.6279,B 16.8368,C -0.1843,E1 16.877,E2 525.4605} C_DIS
LIN {X 34.4098,Y -124.4903,Z 154,A -74.7824,B 16.8368,C -0.1869,E1 16.882,E2 523.6107} C_DIS
LIN {X 37.3436,Y -123.6421,Z 154,A -72.9629,B 16.8365,C -0.2048,E1 16.887,E2 521.7346} C_DIS
LIN {X 41.4106,Y -122.3407,Z 154,A -71.493,B 16.8367,C -0.1918,E1 16.8908,E2 520.3138} C_DIS
LIN {X 45.135,Y -121.0147,Z 154,A -69.8553,B 16.8367,C -0.1898,E1 16.895,E2 518.6882} C_DIS
LIN {X 48.2051,Y -119.8247,Z 154,A -68.5722,B 16.8367,C -0.1854,E1 16.8983,E2 517.4248} C_DIS
LIN {X 52.2336,Y -118.1254,Z 154,A -66.4479,B 16.8367,C -0.1946,E1 16.9038,E2 515.2768} C_DIS
LIN {X 55.2618,Y -116.739,Z 154,A -64.9483,B 16.8367,C -0.1975,E1 16.9076,E2 513.773} C_DIS
LIN {X 58.8638,Y -114.9643,Z 154,A -62.683,B 16.8364,C -0.2176,E1 16.9134,E2 511.448} C_DIS
LIN {X 62.7567,Y -112.8884,Z 154,A -61.1712,B 16.8365,C -0.2047,E1 16.917,E2 509.9875} C_DIS
LIN {X 66.4809,Y -110.7367,Z 154,A -59.2841,B 16.8365,C -0.2072,E1 16.9215,E2 508.1008} C_DIS
LIN {X 69.7437,Y -108.7106,Z 154,A -57.5977,B 16.8365,C -0.2096,E1 16.9255,E2 506.4145} C_DIS
LIN {X 72.9729,Y -106.5699,Z 154,A -55.8845,B 16.8365,C -0.2126,E1 16.9295,E2 504.7} C_DIS
LIN {X 76.1283,Y -104.3398,Z 154,A -54.1197,B 16.8364,C -0.2177,E1 16.9335,E2 502.9271} C_DIS
LIN {X 80.4215,Y -101.067,Z 154,A -51.8043,B 16.8364,C -0.2196,E1 16.9386,E2 500.6183} C_DIS
LIN {X 83.813,Y -98.273,Z 154,A -49.8834,B 16.8364,C -0.2226,E1 16.9427,E2 498.6984} C_DIS
LIN {X 87.0114,Y -95.4529,Z 154,A -48.2036,B 16.8364,C -0.219,E1 16.9462,E2 497.0414} C_DIS
LIN {X 89.001,Y -93.6006,Z 154,A -46.7065,B 16.8362,C -0.2323,E1 16.9493,E2 495.5082} C_DIS
LIN {X 92.3639,Y -90.2835,Z 154,A -44.6757,B 16.8362,C -0.2347,E1 16.9533,E2 493.4823} C_DIS
LIN {X 95.273,Y -87.2082,Z 154,A -43.0001,B 16.8362,C -0.2317,E1 16.9564,E2 491.8283} C_DIS
LIN {X 97.5693,Y -84.6314,Z 154,A -41.2598,B 16.836,C -0.2431,E1 16.9597,E2 490.0611} C_DIS
LIN {X 100.4162,Y -81.2329,Z 154,A -39.3341,B 16.836,C -0.2464,E1 16.9631,E2 488.1377} C_DIS
LIN {X 103.0192,Y -77.9052,Z 154,A -37.5578,B 16.836,C -0.2475,E1 16.9661,E2 486.3704} C_DIS
LIN {X 105.5743,Y -74.4058,Z 154,A -35.5768,B 16.8359,C -0.2547,E1 16.9693,E2 484.3798} C_DIS
LIN {X 108.0561,Y -70.7541,Z 154,A -33.6456,B 16.8359,C -0.2588,E1 16.9723,E2 482.4492} C_DIS
LIN {X 110.1476,Y -67.4513,Z 154,A -31.9104,B 16.8357,C -0.2635,E1 16.9749,E2 480.7115} C_DIS
LIN {X 112.366,Y -63.688,Z 154,A -30.0539,B 16.8357,C -0.2658,E1 16.9775,E2 478.862} C_DIS
LIN {X 114.0531,Y -60.6131,Z 154,A -28.6209,B 16.8357,C -0.2655,E1 16.9794,E2 477.4413} C_DIS
LIN {X 116.0742,Y -56.6456,Z 154,A -26.5087,B 16.8355,C -0.2761,E1 16.982,E2 475.3101} C_DIS
LIN {X 117.7569,Y -53.0575,Z 154,A -24.8281,B 16.8355,C -0.2783,E1 16.984,E2 473.6362} C_DIS
LIN {X 119.1519,Y -49.8448,Z 154,A -23.3111,B 16.8355,C -0.2814,E1 16.9856,E2 472.1213} C_DIS
LIN {X 121.5208,Y -43.7536,Z 154,A -20.4531,B 16.8353,C -0.2883,E1 16.9885,E2 469.2641} C_DIS
LIN {X 122.5674,Y -40.7301,Z 154,A -19.0543,B 16.8353,C -0.2917,E1 16.9897,E2 467.8658} C_DIS
LIN {X 123.4333,Y -38.0258,Z 154,A -17.5487,B 16.8351,C -0.3046,E1 16.991,E2 466.3292} C_DIS
LIN {X 124.7271,Y -33.5398,Z 154,A -15.8999,B 16.8352,C -0.295,E1 16.9922,E2 464.7276} C_DIS
LIN {X 125.5678,Y -30.2398,Z 154,A -14.211,B 16.835,C -0.3062,E1 16.9934,E2 463.0155} C_DIS
LIN {X 126.1764,Y -27.5929,Z 154,A -12.8535,B 16.8349,C -0.3155,E1 16.9942,E2 461.6382} C_DIS
LIN {X 127.0668,Y -23.15,Z 154,A -11.2098,B 16.835,C -0.308,E1 16.9951,E2 460.0352} C_DIS
LIN {X 127.8424,Y -18.3869,Z 154,A -8.8878,B 16.8348,C -0.3212,E1 16.9961,E2 457.6888} C_DIS
LIN {X 128.3427,Y -14.5045,Z 154,A -6.8669,B 16.8345,C -0.3371,E1 16.9968,E2 455.6318} C_DIS
LIN {X 128.6669,Y -11.2589,Z 154,A -5.2982,B 16.8343,C -0.3462,E1 16.9971,E2 454.0465} C_DIS
LIN {X 128.9617,Y -7.1481,Z 154,A -3.8465,B 16.8344,C -0.3376,E1 16.9974,E2 452.6372} C_DIS
LIN {X 129.1043,Y -3.7268,Z 154,A -2.4106,B 16.8344,C -0.3392,E1 16.9974,E2 451.2091} C_DIS
LIN {X 129.1595,Y 0.342,Z 154,A -0.5622,B 16.8343,C -0.3463,E1 16.9975,E2 449.3532} C_DIS
LIN {X 128.8675,Y 8.6874,Z 154,A 2.9637,B 16.8342,C -0.3509,E1 16.9971,E2 445.8437} C_DIS
LIN {X 128.3412,Y 14.5128,Z 154,A 5.5097,B 16.8341,C -0.357,E1 16.9964,E2 443.3002} C_DIS
LIN {X 127.4808,Y 20.7521,Z 154,A 8.4056,B 16.8338,C -0.3691,E1 16.9953,E2 440.3889} C_DIS
LIN {X 126.8791,Y 24.1543,Z 154,A 9.8178,B 16.8338,C -0.3692,E1 16.9946,E2 438.9891} C_DIS
LIN {X 126.3824,Y 26.6386,Z 154,A 11.3859,B 16.8334,C -0.3891,E1 16.9936,E2 437.3671} C_DIS
LIN {X 125.5854,Y 30.1668,Z 154,A 12.6683,B 16.8335,C -0.3818,E1 16.9928,E2 436.1209} C_DIS
LIN {X 124.5148,Y 34.3219,Z 154,A 14.4823,B 16.8335,C -0.3841,E1 16.9915,E2 434.3153} C_DIS
LIN {X 123.5032,Y 37.7977,Z 154,A 16.0999,B 16.8334,C -0.3891,E1 16.9902,E2 432.6944} C_DIS
LIN {X 122.165,Y 41.9233,Z 154,A 17.9203,B 16.8334,C -0.3908,E1 16.9886,E2 430.8842} C_DIS
LIN {X 121.0496,Y 45.0416,Z 154,A 19.327,B 16.8333,C -0.3927,E1 16.9873,E2 429.4832} C_DIS
LIN {X 119.8701,Y 48.0923,Z 154,A 20.6061,B 16.8333,C -0.3904,E1 16.986,E2 428.2227} C_DIS
LIN {X 118.159,Y 52.1585,Z 154,A 22.7127,B 16.8331,C -0.4013,E1 16.9837,E2 426.0966} C_DIS
LIN {X 115.4236,Y 57.9617,Z 154,A 25.7604,B 16.8327,C -0.4163,E1 16.98,E2 423.0226} C_DIS
LIN {X 113.511,Y 61.6236,Z 154,A 27.5292,B 16.8327,C -0.4188,E1 16.9776,E2 421.2596} C_DIS
LIN {X 111.4008,Y 65.3608,Z 154,A 29.3748,B 16.8327,C -0.4216,E1 16.9751,E2 419.4191} C_DIS
LIN {X 108.7866,Y 69.625,Z 154,A 31.334,B 16.8327,C -0.4178,E1 16.9722,E2 417.4883} C_DIS
LIN {X 104.3169,Y 76.1596,Z 154,A 35.1163,B 16.8323,C -0.4361,E1 16.9662,E2 413.6719} C_DIS
LIN {X 101.7117,Y 79.6049,Z 154,A 36.9941,B 16.8322,C -0.4392,E1 16.963,E2 411.7971} C_DIS
LIN {X 99.0948,Y 82.8398,Z 154,A 38.8431,B 16.8321,C -0.4435,E1 16.9597,E2 409.9464} C_DIS
LIN {X 96.312,Y 86.0591,Z 154,A 40.7094,B 16.832,C -0.4469,E1 16.9563,E2 408.0813} C_DIS
LIN {X 93.4675,Y 89.1403,Z 154,A 42.5665,B 16.8319,C -0.4508,E1 16.9527,E2 406.2234} C_DIS
LIN {X 90.2685,Y 92.3786,Z 154,A 44.301,B 16.832,C -0.4448,E1 16.9493,E2 404.5209} C_DIS
LIN {X 87.8998,Y 94.6351,Z 154,A 45.9835,B 16.8317,C -0.456,E1 16.9459,E2 402.8107} C_DIS
LIN {X 84.7772,Y 97.4424,Z 154,A 47.7902,B 16.8317,C -0.4576,E1 16.9421,E2 401.0096} C_DIS
LIN {X 81.7334,Y 100.009,Z 154,A 49.614,B 16.8316,C -0.4629,E1 16.9382,E2 399.1781} C_DIS
LIN {X 78.2001,Y 102.796,Z 154,A 51.6306,B 16.8314,C -0.4672,E1 16.9337,E2 397.1583} C_DIS
LIN {X 74.7363,Y 105.3412,Z 154,A 53.5091,B 16.8314,C -0.4694,E1 16.9295,E2 395.2825} C_DIS
LIN {X 71.2508,Y 107.7291,Z 154,A 55.6079,B 16.8311,C -0.4803,E1 16.9245,E2 393.1568} C_DIS
LIN {X 68.4259,Y 109.5449,Z 154,A 58.0991,B 16.83,C -0.5183,E1 16.9183,E2 390.547} C_DIS
LIN {X 61.1022,Y 113.7923,Z 154,A 60.643,B 16.8311,C -0.4804,E1 16.9124,E2 388.1451} C_DIS
LIN {X 57.7018,Y 115.5532,Z 154,A 62.2654,B 16.8311,C -0.4799,E1 16.9084,E2 386.5313} C_DIS
LIN {X 54.4242,Y 117.1312,Z 154,A 63.6404,B 16.8313,C -0.4735,E1 16.905,E2 385.1837} C_DIS
LIN {X 50.6144,Y 118.829,Z 154,A 66.3775,B 16.8303,C -0.5065,E1 16.8977,E2 382.3433} C_DIS
LIN {X 45.6615,Y 120.8174,Z 154,A 68.369,B 16.8306,C -0.4957,E1 16.8926,E2 380.3956} C_DIS
LIN {X 42.3743,Y 122.0086,Z 154,A 69.5125,B 16.831,C -0.483,E1 16.8898,E2 379.2994} C_DIS
LIN {X 39.4228,Y 122.9941,Z 154,A 70.8081,B 16.831,C -0.4812,E1 16.8863,E2 378.0138} C_DIS
LIN {X 36.8145,Y 123.801,Z 154,A 72.1708,B 16.8309,C -0.4874,E1 16.8827,E2 376.6337} C_DIS
LIN {X 33.4785,Y 124.7435,Z 154,A 73.7136,B 16.8309,C -0.4886,E1 16.8785,E2 375.0905} C_DIS
LIN {X 29.8038,Y 125.6729,Z 154,A 75.4445,B 16.8308,C -0.4913,E1 16.8738,E2 373.3541} C_DIS
LIN {X 25.9133,Y 126.5316,Z 154,A 77.1251,B 16.8308,C -0.4893,E1 16.8692,E2 371.6839} C_DIS
LIN {X 23.0481,Y 127.0851,Z 154,A 78.6305,B 16.8306,C -0.4971,E1 16.865,E2 370.1544} C_DIS
LIN {X 18.4536,Y 127.8329,Z 154,A 80.4798,B 16.8308,C -0.4905,E1 16.86,E2 368.3306} C_DIS
LIN {X 15.5884,Y 128.2141,Z 154,A 81.908,B 16.8306,C -0.4957,E1 16.856,E2 366.886} C_DIS
LIN {X 11.7587,Y 128.6229,Z 154,A 84.0119,B 16.8303,C -0.5094,E1 16.85,E2 364.7368} C_DIS
LIN {X 7.2576,Y 128.9557,Z 154,A 85.357,B 16.8309,C -0.4874,E1 16.8465,E2 363.4687} C_DIS
LIN {X 0.521,Y 129.1572,Z 154,A 88.0508,B 16.8312,C -0.4774,E1 16.8391,E2 360.8103} C_DIS
LIN {X -5.9897,Y 129.02,Z 154,A 91.303,B 16.8308,C -0.4888,E1 16.8299,E2 357.5182} C_DIS
LIN {X -13.5719,Y 128.4431,Z 154,A 95.1205,B 16.8305,C -0.5022,E1 16.8191,E2 353.6516} C_DIS
LIN {X -17.3112,Y 127.9936,Z 154,A 96.4891,B 16.8308,C -0.4914,E1 16.8154,E2 352.3189} C_DIS
LIN {X -21.0513,Y 127.4309,Z 154,A 98.0619,B 16.8308,C -0.487,E1 16.8111,E2 350.7594} C_DIS
LIN {X -23.6715,Y 126.9714,Z 154,A 99.6534,B 16.8305,C -0.4997,E1 16.8066,E2 349.1213} C_DIS
LIN {X -27.1908,Y 126.2632,Z 154,A 100.914,B 16.8309,C -0.4876,E1 16.8033,E2 347.9002} C_DIS
LIN {X -30.2798,Y 125.5581,Z 154,A 102.3391,B 16.8309,C -0.4871,E1 16.7994,E2 346.4739} C_DIS
LIN {X -34.7098,Y 124.4064,Z 154,A 104.3371,B 16.8309,C -0.4842,E1 16.794,E2 344.4814} C_DIS
LIN {X -38.1938,Y 123.3819,Z 154,A 105.9135,B 16.8311,C -0.4815,E1 16.7898,E2 342.9103} C_DIS
LIN {X -42.2642,Y 122.0468,Z 154,A 107.8115,B 16.8311,C -0.4793,E1 16.7848,E2 341.0142} C_DIS
LIN {X -45.3301,Y 120.9416,Z 154,A 109.2813,B 16.8311,C -0.4784,E1 16.781,E2 339.5429} C_DIS
LIN {X -50.5279,Y 118.8664,Z 154,A 111.7553,B 16.8312,C -0.475,E1 16.7746,E2 337.0724} C_DIS
LIN {X -53.5448,Y 117.5378,Z 154,A 113.3007,B 16.8312,C -0.4757,E1 16.7706,E2 335.5189} C_DIS
LIN {X -56.7561,Y 116.0197,Z 154,A 114.8645,B 16.8312,C -0.4731,E1 16.7667,E2 333.958} C_DIS
LIN {X -59.8753,Y 114.4405,Z 154,A 116.3812,B 16.8314,C -0.4696,E1 16.7629,E2 332.4468} C_DIS
LIN {X -63.4983,Y 112.473,Z 154,A 118.3169,B 16.8314,C -0.4701,E1 16.7582,E2 330.5009} C_DIS
LIN {X -67.2599,Y 110.265,Z 154,A 120.0372,B 16.8316,C -0.4601,E1 16.7541,E2 328.8073} C_DIS
LIN {X -70.8643,Y 107.9835,Z 154,A 122.1457,B 16.8316,C -0.4636,E1 16.7491,E2 326.6761} C_DIS
LIN {X -74.2457,Y 105.6872,Z 154,A 123.9984,B 16.8316,C -0.4615,E1 16.7449,E2 324.821} C_DIS
LIN {X -78.0374,Y 102.9194,Z 154,A 126.076,B 16.8317,C -0.4574,E1 16.7402,E2 322.7464} C_DIS
LIN {X -81.4488,Y 100.2416,Z 154,A 128.0395,B 16.8317,C -0.4548,E1 16.7359,E2 320.7807} C_DIS
LIN {X -84.7395,Y 97.4753,Z 154,A 129.9178,B 16.8319,C -0.4499,E1 16.7319,E2 318.9081} C_DIS
LIN {X -87.9047,Y 94.6305,Z 154,A 131.8283,B 16.8319,C -0.4466,E1 16.728,E2 316.9973} C_DIS
LIN {X -91.0422,Y 91.6159,Z 154,A 133.7249,B 16.8321,C -0.4412,E1 16.7242,E2 315.107} C_DIS
LIN {X -93.814,Y 88.7757,Z 154,A 135.5518,B 16.8321,C -0.4393,E1 16.7207,E2 313.2747} C_DIS
LIN {X -96.853,Y 85.4497,Z 154,A 137.5382,B 16.8323,C -0.4342,E1 16.717,E2 311.2923} C_DIS
LIN {X -99.7347,Y 82.0689,Z 154,A 139.5683,B 16.8323,C -0.4313,E1 16.7133,E2 309.2581} C_DIS
LIN {X -102.4537,Y 78.6476,Z 154,A 141.5078,B 16.8325,C -0.4265,E1 16.71,E2 307.321} C_DIS
LIN {X -105.1089,Y 75.0619,Z 154,A 143.4257,B 16.8327,C -0.4196,E1 16.7069,E2 305.4129} C_DIS
LIN {X -107.4112,Y 71.7286,Z 154,A 145.2473,B 16.8327,C -0.4157,E1 16.704,E2 303.5909} C_DIS
LIN {X -109.2265,Y 68.9327,Z 154,A 147.3023,B 16.8324,C -0.4295,E1 16.7009,E2 301.4715} C_DIS
LIN {X -111.6654,Y 64.908,Z 154,A 148.8993,B 16.8329,C -0.4087,E1 16.6987,E2 299.9341} C_DIS
LIN {X -113.4955,Y 61.6522,Z 154,A 150.792,B 16.8329,C -0.4115,E1 16.6961,E2 298.0166} C_DIS
LIN {X -115.5496,Y 57.709,Z 154,A 153.0423,B 16.8328,C -0.4145,E1 16.6933,E2 295.7368} C_DIS
LIN {X -117.5284,Y 53.5652,Z 154,A 154.5294,B 16.8333,C -0.3919,E1 16.6916,E2 294.3162} C_DIS
LIN {X -119.0625,Y 50.0587,Z 154,A 156.2356,B 16.8334,C -0.3873,E1 16.6897,E2 292.6114} C_DIS
LIN {X -120.3073,Y 46.988,Z 154,A 157.692,B 16.8335,C -0.3826,E1 16.6882,E2 291.1586} C_DIS
LIN {X -121.4458,Y 43.9615,Z 154,A 159.1512,B 16.8335,C -0.3792,E1 16.6868,E2 289.6985} C_DIS
LIN {X -122.7749,Y 40.1051,Z 154,A 161.2487,B 16.8335,C -0.3827,E1 16.6849,E2 287.5705} C_DIS
LIN {X -124.2535,Y 35.2563,Z 154,A 163.3176,B 16.8338,C -0.3705,E1 16.6833,E2 285.5254} C_DIS
LIN {X -125.2422,Y 31.5617,Z 154,A 165.0037,B 16.8338,C -0.3651,E1 16.6821,E2 283.843} C_DIS
LIN {X -126.1549,Y 27.6922,Z 154,A 166.8068,B 16.834,C -0.361,E1 16.681,E2 282.0378} C_DIS
LIN {X -126.7252,Y 24.9596,Z 154,A 168.1126,B 16.834,C -0.3593,E1 16.6803,E2 280.726} C_DIS
LIN {X -127.3942,Y 21.271,Z 154,A 169.5783,B 16.8342,C -0.3483,E1 16.6796,E2 279.2852} C_DIS
LIN {X -127.8841,Y 18.0951,Z 154,A 171.1178,B 16.8342,C -0.3474,E1 16.679,E2 277.7347} C_DIS
LIN {X -128.3537,Y 14.4024,Z 154,A 172.9265,B 16.8342,C -0.3472,E1 16.6784,E2 275.9101} C_DIS
LIN {X -128.7543,Y 10.224,Z 154,A 174.8415,B 16.8343,C -0.3431,E1 16.6779,E2 273.9916} C_DIS
LIN {X -129.032,Y 5.749,Z 154,A 176.7017,B 16.8345,C -0.3331,E1 16.6776,E2 272.149} C_DIS
LIN {X -129.1522,Y 1.3952,Z 154,A 178.6739,B 16.8346,C -0.3284,E1 16.6776,E2 270.1747} C_DIS
LIN {X -129.135,Y -2.4621,Z 154,A -179.4851,B 16.8346,C -0.3271,E1 16.6776,E2 268.3209} C_DIS
LIN {X -128.9588,Y -7.206,Z 154,A -177.4497,B 16.8348,C -0.3185,E1 16.6779,E2 266.2964} C_DIS
LIN {X -128.7031,Y -10.8305,Z 154,A -175.8466,B 16.8349,C -0.3134,E1 16.6782,E2 264.6963} C_DIS
LIN {X -128.4016,Y -13.9573,Z 154,A -174.4709,B 16.8349,C -0.3087,E1 16.6786,E2 263.3245} C_DIS
LIN {X -127.8977,Y -18.0002,Z 154,A -172.6374,B 16.8351,C -0.304,E1 16.6793,E2 261.4902} C_DIS
LIN {X -127.4437,Y -20.9743,Z 154,A -171.2527,B 16.8351,C -0.3015,E1 16.6799,E2 260.1014} C_DIS
LIN {X -126.7525,Y -24.8166,Z 154,A -169.4418,B 16.8351,C -0.2988,E1 16.6808,E2 258.2835} C_DIS
LIN {X -125.9172,Y -28.7501,Z 154,A -167.7378,B 16.8353,C -0.2911,E1 16.6819,E2 256.5908} C_DIS
LIN {X -124.9146,Y -32.837,Z 154,A -165.8167,B 16.8353,C -0.2873,E1 16.6832,E2 254.6657} C_DIS
LIN {X -124.0463,Y -35.9768,Z 154,A -164.3708,B 16.8354,C -0.2831,E1 16.6843,E2 253.2213} C_DIS
LIN {X -122.7972,Y -40.0392,Z 154,A -162.1631,B 16.8354,C -0.2877,E1 16.6862,E2 250.9783} C_DIS
LIN {X -121.7006,Y -43.255,Z 154,A -160.9277,B 16.8356,C -0.275,E1 16.6873,E2 249.7762} C_DIS
LIN {X -120.5005,Y -46.4909,Z 154,A -159.4302,B 16.8356,C -0.2697,E1 16.6888,E2 248.2841} C_DIS
LIN {X -119.2423,Y -49.6283,Z 154,A -158.1187,B 16.8358,C -0.2597,E1 16.6901,E2 246.996} C_DIS
LIN {X -118.1607,Y -52.1548,Z 154,A -156.5691,B 16.8357,C -0.2666,E1 16.6919,E2 245.4093} C_DIS
LIN {X -116.3369,Y -56.1035,Z 154,A -154.6337,B 16.8357,C -0.2616,E1 16.6942,E2 243.4751} C_DIS
LIN {X -114.4785,Y -59.803,Z 154,A -152.9667,B 16.8359,C -0.2514,E1 16.6963,E2 241.8297} C_DIS
LIN {X -112.5191,Y -63.4164,Z 154,A -151.0846,B 16.8359,C -0.2485,E1 16.6989,E2 239.9425} C_DIS
LIN {X -110.9169,Y -66.1785,Z 154,A -149.6446,B 16.8359,C -0.2456,E1 16.7009,E2 238.501} C_DIS
LIN {X -109.1108,Y -69.1162,Z 154,A -148.0174,B 16.836,C -0.2448,E1 16.7033,E2 236.8638} C_DIS
LIN {X -107.3851,Y -71.7677,Z 154,A -146.5767,B 16.836,C -0.2425,E1 16.7056,E2 235.42} C_DIS
LIN {X -104.9017,Y -75.3517,Z 154,A -144.6783,B 16.8361,C -0.2367,E1 16.7086,E2 233.5273} C_DIS
LIN {X -102.2292,Y -78.9392,Z 154,A -142.1398,B 16.8359,C -0.2496,E1 16.713,E2 230.9253} C_DIS
LIN {X -99.2677,Y -82.6328,Z 154,A -140.5161,B 16.8362,C -0.2298,E1 16.7158,E2 229.3591} C_DIS
LIN {X -96.531,Y -85.8141,Z 154,A -138.6397,B 16.8362,C -0.2261,E1 16.7193,E2 227.4823} C_DIS
LIN {X -94.3461,Y -88.2101,Z 154,A -137.215,B 16.8363,C -0.2226,E1 16.722,E2 226.06} C_DIS
LIN {X -92.1068,Y -90.5456,Z 154,A -135.8617,B 16.8363,C -0.2171,E1 16.7246,E2 224.7172} C_DIS
LIN {X -86.2182,Y -96.1695,Z 154,A -132.1406,B 16.8364,C -0.2133,E1 16.7322,E2 220.9856} C_DIS
LIN {X -82.7845,Y -99.1411,Z 154,A -130.2334,B 16.8365,C -0.2061,E1 16.7362,E2 219.092} C_DIS
LIN {X -79.1879,Y -102.0365,Z 154,A -128.1219,B 16.8365,C -0.2045,E1 16.7408,E2 216.974} C_DIS
LIN {X -76.0733,Y -104.3797,Z 154,A -126.3318,B 16.8365,C -0.2036,E1 16.7449,E2 215.1774} C_DIS
LIN {X -71.7219,Y -107.4157,Z 154,A -123.9634,B 16.8365,C -0.2003,E1 16.7503,E2 212.8081} C_DIS
LIN {X -67.81,Y -109.9276,Z 154,A -121.3376,B 16.8364,C -0.2157,E1 16.7567,E2 210.1164} C_DIS
LIN {X -63.6258,Y -112.4014,Z 154,A -119.7018,B 16.8366,C -0.1956,E1 16.7605,E2 208.5427} C_DIS
LIN {X -60.6979,Y -114.0086,Z 154,A -118.3573,B 16.8367,C -0.1892,E1 16.7638,E2 207.2146} C_DIS
LIN {X -57.6678,Y -115.57,Z 154,A -116.7657,B 16.8367,C -0.1899,E1 16.7678,E2 205.6139} C_DIS
LIN {X -53.4175,Y -117.5959,Z 154,A -114.7386,B 16.8367,C -0.1855,E1 16.7729,E2 203.5944} C_DIS
LIN {X -48.64,Y -119.6494,Z 154,A -112.0139,B 16.8367,C -0.197,E1 16.78,E2 200.8204} C_DIS
LIN {X -45.3631,Y -120.9292,Z 154,A -110.8531,B 16.8367,C -0.1822,E1 16.7829,E2 199.7068} C_DIS
LIN {X -42.2317,Y -122.0581,Z 154,A -109.3514,B 16.8367,C -0.1818,E1 16.7869,E2 198.2022} C_DIS
LIN {X -39.2232,Y -123.0579,Z 154,A -107.8388,B 16.8367,C -0.1842,E1 16.7909,E2 196.6769} C_DIS
LIN {X -35.1727,Y -124.2769,Z 154,A -106.0424,B 16.8367,C -0.1802,E1 16.7957,E2 194.8899} C_DIS
LIN {X -31.7655,Y -125.1905,Z 154,A -104.4104,B 16.8367,C -0.1815,E1 16.8002,E2 193.2497} C_DIS
LIN {X -27.8085,Y -126.1298,Z 154,A -102.7295,B 16.8368,C -0.1764,E1 16.8047,E2 191.5831} C_DIS
LIN {X -23.1828,Y -127.0609,Z 154,A -100.5408,B 16.8368,C -0.1788,E1 16.8107,E2 189.3826} C_DIS
LIN {X -16.4473,Y -128.1068,Z 154,A -97.3602,B 16.8368,C -0.1832,E1 16.8196,E2 186.1827} C_DIS
LIN {X -11.5384,Y -128.6433,Z 154,A -95.2514,B 16.8368,C -0.1801,E1 16.8254,E2 184.0828} C_DIS
LIN {X -7.5817,Y -128.9358,Z 154,A -93.5783,B 16.8368,C -0.1771,E1 16.83,E2 182.4193} C_DIS
LIN {X -3.3684,Y -129.1143,Z 154,A -91.6568,B 16.8368,C -0.179,E1 16.8354,E2 180.4909} C_DIS
LIN {X 0.9058,Y -129.1537,Z 154,A -89.8866,B 16.8368,C -0.175,E1 16.8403,E2 178.7346} C_DIS
Enddeposition()
LIN {X 0.9058,Y -129.1537,Z 154,A -89.8866,B 16.8368,C -0.175,E1 16.8403,E2 178.7346} C_DIS
Startdeposition()
$VEL.CP = VEL_PRINT
LIN {X -0.6637,Y -128.2187,Z 154,A -91.2527,B 16.837,C -0.163,E1 16.8365,E2 180.142} C_DIS
LIN {X -4.7189,Y -128.1338,Z 154,A -93.0348,B 16.837,C -0.1639,E1 16.8315,E2 181.9214} C_DIS
LIN {X -7.8595,Y -127.9792,Z 154,A -94.5055,B 16.837,C -0.1617,E1 16.8274,E2 183.4003} C_DIS
LIN {X -12.0226,Y -127.6556,Z 154,A -96.4054,B 16.837,C -0.1607,E1 16.8221,E2 185.3048} C_DIS
LIN {X -15.7436,Y -127.2512,Z 154,A -97.9587,B 16.837,C -0.165,E1 16.8178,E2 186.8449} C_DIS
LIN {X -18.8404,Y -126.8304,Z 154,A -99.3656,B 16.837,C -0.165,E1 16.8139,E2 188.2535} C_DIS
LIN {X -21.9268,Y -126.3332,Z 154,A -100.939,B 16.837,C -0.1596,E1 16.8095,E2 189.8476} C_DIS
LIN {X -25.9316,Y -125.571,Z 154,A -102.7175,B 16.837,C -0.1619,E1 16.8047,E2 191.6215} C_DIS
LIN {X -29.6357,Y -124.7489,Z 154,A -104.294,B 16.837,C -0.1667,E1 16.8004,E2 193.1846} C_DIS
LIN {X -33.0779,Y -123.8799,Z 154,A -105.9634,B 16.837,C -0.1649,E1 16.7959,E2 194.8637} C_DIS
LIN {X -37.2173,Y -122.7002,Z 154,A -107.8046,B 16.837,C -0.1689,E1 16.791,E2 196.6956} C_DIS
LIN {X -41.0883,Y -121.4598,Z 154,A -109.7873,B 16.837,C -0.165,E1 16.7857,E2 198.6976} C_DIS
LIN {X -44.726,Y -120.1665,Z 154,A -111.5165,B 16.837,C -0.1664,E1 16.7811,E2 200.4272} C_DIS
LIN {X -48.4987,Y -118.6953,Z 154,A -113.1768,B 16.837,C -0.173,E1 16.7769,E2 202.0704} C_DIS
LIN {X -51.3715,Y -117.4801,Z 154,A -114.5833,B 16.837,C -0.174,E1 16.7732,E2 203.4782} C_DIS
LIN {X -54.8109,Y -115.9152,Z 154,A -116.2669,B 16.837,C -0.1761,E1 16.769,E2 205.1611} C_DIS
LIN {X -57.6513,Y -114.5294,Z 154,A -117.6765,B 16.8369,C -0.1779,E1 16.7654,E2 206.5702} C_DIS
LIN {X -60.4454,Y -113.0807,Z 154,A -119.1801,B 16.8369,C -0.1766,E1 16.7617,E2 208.0847} C_DIS
LIN {X -64.0374,Y -111.086,Z 154,A -121.0625,B 16.8369,C -0.1776,E1 16.7571,E2 209.972} C_DIS
LIN {X -67.2785,Y -109.1535,Z 154,A -122.6369,B 16.8369,C -0.1836,E1 16.7534,E2 211.5331} C_DIS
LIN {X -70.2419,Y -107.2706,Z 154,A -124.3238,B 16.8369,C -0.1822,E1 16.7494,E2 213.2331} C_DIS
LIN {X -73.2975,Y -105.206,Z 154,A -125.8669,B 16.8368,C -0.1882,E1 16.7459,E2 214.7635} C_DIS
LIN {X -75.8539,Y -103.378,Z 154,A -127.4018,B 16.8368,C -0.1864,E1 16.7424,E2 216.3129} C_DIS
LIN {X -78.984,Y -101.007,Z 154,A -129.1801,B 16.8368,C -0.1887,E1 16.7384,E2 218.0932} C_DIS
LIN {X -82.2084,Y -98.4005,Z 154,A -131.0031,B 16.8368,C -0.193,E1 16.7345,E2 219.9119} C_DIS
LIN {X -85.279,Y -95.7519,Z 154,A -132.8421,B 16.8368,C -0.1956,E1 16.7306,E2 221.7531} C_DIS
LIN {X -88.318,Y -92.9563,Z 154,A -134.6392,B 16.8366,C -0.2007,E1 16.727,E2 223.5437} C_DIS
LIN {X -91.2441,Y -90.086,Z 154,A -136.5319,B 16.8366,C -0.2025,E1 16.7232,E2 225.4423} C_DIS
LIN {X -93.9481,Y -87.2616,Z 154,A -138.2727,B 16.8366,C -0.2065,E1 16.7199,E2 227.1813} C_DIS
LIN {X -96.8777,Y -83.9982,Z 154,A -140.2396,B 16.8366,C -0.2105,E1 16.7163,E2 229.1476} C_DIS
LIN {X -99.4243,Y -80.9671,Z 154,A -141.9946,B 16.8365,C -0.2149,E1 16.7131,E2 230.8998} C_DIS
LIN {X -102.0398,Y -77.6453,Z 154,A -143.9869,B 16.8365,C -0.2161,E1 16.7097,E2 232.9025} C_DIS
LIN {X -104.5327,Y -74.2555,Z 154,A -145.8616,B 16.8365,C -0.2208,E1 16.7067,E2 234.775} C_DIS
LIN {X -106.6192,Y -71.2261,Z 154,A -147.3643,B 16.8363,C -0.2291,E1 16.7043,E2 236.2602} C_DIS
LIN {X -108.3312,Y -68.5945,Z 154,A -148.8039,B 16.8363,C -0.2315,E1 16.7021,E2 237.7029} C_DIS
LIN {X -109.9783,Y -65.9219,Z 154,A -150.3565,B 16.8363,C -0.2305,E1 16.6999,E2 239.2713} C_DIS
LIN {X -112.0038,Y -62.4186,Z 154,A -152.0386,B 16.8362,C -0.239,E1 16.6976,E2 240.9374} C_DIS
LIN {X -113.8132,Y -59.0531,Z 154,A -153.7975,B 16.8362,C -0.2419,E1 16.6953,E2 242.7005} C_DIS
LIN {X -115.6324,Y -55.403,Z 154,A -155.6019,B 16.836,C -0.2473,E1 16.6931,E2 244.501} C_DIS
LIN {X -117.2222,Y -51.9565,Z 154,A -157.3176,B 16.836,C -0.2514,E1 16.6911,E2 246.2173} C_DIS
LIN {X -118.4597,Y -49.069,Z 154,A -158.7325,B 16.836,C -0.2549,E1 16.6895,E2 247.632} C_DIS
LIN {X -119.6262,Y -46.152,Z 154,A -160.1476,B 16.8359,C -0.2585,E1 16.6881,E2 249.0468} C_DIS
LIN {X -120.7209,Y -43.2077,Z 154,A -161.5628,B 16.8359,C -0.2621,E1 16.6867,E2 250.4619} C_DIS
LIN {X -121.7427,Y -40.2385,Z 154,A -162.9968,B 16.8358,C -0.2651,E1 16.6855,E2 251.8978} C_DIS
LIN {X -122.9632,Y -36.339,Z 154,A -164.952,B 16.8358,C -0.2665,E1 16.6839,E2 253.8656} C_DIS
LIN {X -124.1654,Y -31.9927,Z 154,A -166.9137,B 16.8356,C -0.274,E1 16.6824,E2 255.8189} C_DIS
LIN {X -125.083,Y -28.1913,Z 154,A -168.7757,B 16.8356,C -0.2757,E1 16.6812,E2 257.6919} C_DIS
LIN {X -125.933,Y -24.1098,Z 154,A -170.5157,B 16.8355,C -0.2849,E1 16.6803,E2 259.4156} C_DIS
LIN {X -126.5941,Y -20.3687,Z 154,A -172.2216,B 16.8354,C -0.2897,E1 16.6795,E2 261.1205} C_DIS
LIN {X -127.1059,Y -16.8688,Z 154,A -173.9044,B 16.8354,C -0.2914,E1 16.6789,E2 262.8128} C_DIS
LIN {X -127.5391,Y -13.209,Z 154,A -175.6212,B 16.8354,C -0.2943,E1 16.6783,E2 264.5354} C_DIS
LIN {X -127.8731,Y -9.4297,Z 154,A -177.1817,B 16.8352,C -0.3035,E1 16.678,E2 266.0785} C_DIS
LIN {X -128.0658,Y -6.2938,Z 154,A -178.591,B 16.8351,C -0.3076,E1 16.6778,E2 267.4866} C_DIS
LIN {X -128.1968,Y -2.4834,Z 154,A 179.5922,B 16.8351,C -0.3094,E1 16.6776,E2 269.3139} C_DIS
LIN {X -128.212,Y 1.5676,Z 154,A 177.6938,B 16.835,C -0.3123,E1 16.6776,E2 271.2199} C_DIS
LIN {X -128.0981,Y 5.634,Z 154,A 176.055,B 16.8348,C -0.3232,E1 16.6778,E2 272.8361} C_DIS
LIN {X -127.9216,Y 8.7656,Z 154,A 174.5796,B 16.8348,C -0.3253,E1 16.6781,E2 274.3179} C_DIS
LIN {X -127.6025,Y 12.5755,Z 154,A 172.8876,B 16.8347,C -0.331,E1 16.6785,E2 276.0058} C_DIS
LIN {X -127.1735,Y 16.3528,Z 154,A 171.1577,B 16.8346,C -0.3352,E1 16.679,E2 277.7368} C_DIS
LIN {X -126.7344,Y 19.4631,Z 154,A 169.744,B 16.8345,C -0.3392,E1 16.6796,E2 279.1497} C_DIS
LIN {X -126.2195,Y 22.562,Z 154,A 168.3291,B 16.8345,C -0.3431,E1 16.6803,E2 280.5639} C_DIS
LIN {X -125.576,Y 25.9074,Z 154,A 166.6676,B 16.8345,C -0.3436,E1 16.6812,E2 282.2389} C_DIS
LIN {X -124.7891,Y 29.4687,Z 154,A 164.9562,B 16.8344,C -0.3461,E1 16.6823,E2 283.9572} C_DIS
LIN {X -123.752,Y 33.5575,Z 154,A 163.0944,B 16.8342,C -0.3524,E1 16.6836,E2 285.8138} C_DIS
LIN {X -122.4347,Y 38.0849,Z 154,A 160.8884,B 16.8342,C -0.3557,E1 16.6854,E2 288.028} C_DIS
LIN {X -121.0851,Y 42.1755,Z 154,A 159.121,B 16.8339,C -0.366,E1 16.687,E2 289.7749} C_DIS
LIN {X -119.9504,Y 45.3031,Z 154,A 157.6482,B 16.8339,C -0.3708,E1 16.6884,E2 291.2441} C_DIS
LIN {X -118.7087,Y 48.4655,Z 154,A 156.1399,B 16.8337,C -0.3754,E1 16.6899,E2 292.7492} C_DIS
LIN {X -117.4854,Y 51.3592,Z 154,A 154.6157,B 16.8337,C -0.3758,E1 16.6916,E2 294.2849} C_DIS
LIN {X -115.8871,Y 54.8698,Z 154,A 152.995,B 16.8336,C -0.3838,E1 16.6935,E2 295.8916} C_DIS
LIN {X -114.5144,Y 57.6808,Z 154,A 151.5875,B 16.8335,C -0.3874,E1 16.6953,E2 297.2982} C_DIS
LIN {X -113.0727,Y 60.4603,Z 154,A 150.0396,B 16.8335,C -0.3868,E1 16.6973,E2 298.861} C_DIS
LIN {X -111.1134,Y 63.9899,Z 154,A 148.2164,B 16.8334,C -0.3911,E1 16.6998,E2 300.6839} C_DIS
LIN {X -108.9077,Y 67.6753,Z 154,A 146.3315,B 16.8333,C -0.3973,E1 16.7025,E2 302.5622} C_DIS
LIN {X -106.9781,Y 70.6862,Z 154,A 144.7972,B 16.8331,C -0.4034,E1 16.7049,E2 304.0872} C_DIS
LIN {X -104.957,Y 73.6542,Z 154,A 143.036,B 16.8331,C -0.4028,E1 16.7077,E2 305.8638} C_DIS
LIN {X -102.4386,Y 77.1179,Z 154,A 141.1335,B 16.8331,C -0.408,E1 16.7108,E2 307.7624} C_DIS
LIN {X -99.9011,Y 80.3779,Z 154,A 139.3042,B 16.8329,C -0.4131,E1 16.714,E2 309.5873} C_DIS
LIN {X -97.3087,Y 83.4978,Z 154,A 137.4922,B 16.8328,C -0.4175,E1 16.7173,E2 311.3969} C_DIS
LIN {X -94.6651,Y 86.484,Z 154,A 135.6149,B 16.8328,C -0.4188,E1 16.7208,E2 313.2825} C_DIS
LIN {X -91.7725,Y 89.5473,Z 154,A 133.799,B 16.8326,C -0.4251,E1 16.7243,E2 315.0886} C_DIS
LIN {X -88.8528,Y 92.4453,Z 154,A 131.8909,B 16.8326,C -0.4271,E1 16.7281,E2 317.0022} C_DIS
LIN {X -85.7656,Y 95.3161,Z 154,A 129.9762,B 16.8325,C -0.4302,E1 16.732,E2 318.9179} C_DIS
LIN {X -82.5537,Y 98.1108,Z 154,A 128.1216,B 16.8323,C -0.4356,E1 16.736,E2 320.7648} C_DIS
LIN {X -79.5096,Y 100.5942,Z 154,A 126.2816,B 16.8323,C -0.4365,E1 16.74,E2 322.6122} C_DIS
LIN {X -75.7264,Y 103.4716,Z 154,A 124.1524,B 16.8323,C -0.4404,E1 16.7447,E2 324.7395} C_DIS
LIN {X -72.5408,Y 105.7291,Z 154,A 122.427,B 16.8321,C -0.4442,E1 16.7487,E2 326.4607} C_DIS
LIN {X -69.1326,Y 107.9884,Z 154,A 120.7454,B 16.8319,C -0.452,E1 16.7526,E2 328.1239} C_DIS
LIN {X -65.9135,Y 109.9833,Z 154,A 118.8794,B 16.8319,C -0.4494,E1 16.7571,E2 330.0075} C_DIS
LIN {X -62.3824,Y 112.0239,Z 154,A 117.1909,B 16.8318,C -0.4565,E1 16.7611,E2 331.6791} C_DIS
LIN {X -59.8501,Y 113.3946,Z 154,A 115.8339,B 16.8318,C -0.4563,E1 16.7645,E2 333.0426} C_DIS
LIN {X -56.8269,Y 114.9392,Z 154,A 114.386,B 16.8317,C -0.4607,E1 16.7681,E2 334.4811} C_DIS
LIN {X -53.9949,Y 116.2967,Z 154,A 112.839,B 16.8317,C -0.4582,E1 16.772,E2 336.0428} C_DIS
LIN {X -50.5247,Y 117.8462,Z 154,A 111.2511,B 16.8317,C -0.4639,E1 16.776,E2 337.6168} C_DIS
LIN {X -47.6221,Y 119.0486,Z 154,A 109.8408,B 16.8316,C -0.4655,E1 16.7797,E2 339.0264} C_DIS
LIN {X -44.6741,Y 120.186,Z 154,A 108.4256,B 16.8316,C -0.4671,E1 16.7834,E2 340.4407} C_DIS
LIN {X -41.6992,Y 121.2503,Z 154,A 107.0101,B 16.8315,C -0.4685,E1 16.7871,E2 341.8553} C_DIS
LIN {X -38.0841,Y 122.4349,Z 154,A 105.1028,B 16.8316,C -0.4637,E1 16.7922,E2 343.7845} C_DIS
LIN {X -34.1966,Y 123.5762,Z 154,A 103.3714,B 16.8315,C -0.468,E1 16.7969,E2 345.5055} C_DIS
LIN {X -30.257,Y 124.5991,Z 154,A 101.5495,B 16.8315,C -0.4694,E1 16.8018,E2 347.3263} C_DIS
LIN {X -25.884,Y 125.5807,Z 154,A 99.5962,B 16.8314,C -0.4725,E1 16.8071,E2 349.2726} C_DIS
LIN {X -22.5647,Y 126.219,Z 154,A 98.1447,B 16.8313,C -0.4754,E1 16.8111,E2 350.7164} C_DIS
LIN {X -19.4666,Y 126.7339,Z 154,A 96.7422,B 16.8313,C -0.4763,E1 16.8149,E2 352.1178} C_DIS
LIN {X -16.3636,Y 127.1721,Z 154,A 95.3438,B 16.8313,C -0.4771,E1 16.8188,E2 353.5151} C_DIS
LIN {X -12.5151,Y 127.6083,Z 154,A 93.6699,B 16.8312,C -0.4797,E1 16.8234,E2 355.1815} C_DIS
LIN {X -9.3481,Y 127.8791,Z 154,A 92.1113,B 16.8312,C -0.4757,E1 16.8278,E2 356.7549} C_DIS
LIN {X -5.3344,Y 128.1098,Z 154,A 90.3507,B 16.8312,C -0.4773,E1 16.8327,E2 358.5105} C_DIS
LIN {X -1.5318,Y 128.2126,Z 154,A 88.7107,B 16.8312,C -0.4796,E1 16.8373,E2 360.1429} C_DIS
LIN {X 1.6297,Y 128.211,Z 154,A 87.2574,B 16.8312,C -0.4784,E1 16.8413,E2 361.6001} C_DIS
LIN {X 5.6507,Y 128.0974,Z 154,A 85.4984,B 16.8312,C -0.4796,E1 16.8462,E2 363.354} C_DIS
LIN {X 8.8497,Y 127.9154,Z 154,A 84.031,B 16.8312,C -0.4784,E1 16.8503,E2 364.8248} C_DIS
LIN {X 11.957,Y 127.6618,Z 154,A 82.5272,B 16.8313,C -0.4745,E1 16.8545,E2 366.3406} C_DIS
LIN {X 15.7124,Y 127.2549,Z 154,A 80.9718,B 16.8313,C -0.4785,E1 16.8588,E2 367.8805} C_DIS
LIN {X 18.5912,Y 126.866,Z 154,A 79.6554,B 16.8313,C -0.4775,E1 16.8625,E2 369.1986} C_DIS
LIN {X 21.9405,Y 126.3307,Z 154,A 77.9777,B 16.8313,C -0.4715,E1 16.8671,E2 370.8942} C_DIS
LIN {X 25.9248,Y 125.5724,Z 154,A 76.2146,B 16.8313,C -0.4723,E1 16.8719,E2 372.6513} C_DIS
LIN {X 29.6305,Y 124.7501,Z 154,A 74.5032,B 16.8314,C -0.4708,E1 16.8766,E2 374.3642} C_DIS
LIN {X 33.5596,Y 123.7514,Z 154,A 72.6892,B 16.8314,C -0.4695,E1 16.8815,E2 376.1782} C_DIS
LIN {X 37.2215,Y 122.6989,Z 154,A 71.1649,B 16.8314,C -0.4742,E1 16.8855,E2 377.6822} C_DIS
LIN {X 40.7273,Y 121.58,Z 154,A 69.4434,B 16.8314,C -0.4702,E1 16.8901,E2 379.4124} C_DIS
LIN {X 44.7167,Y 120.17,Z 154,A 67.4558,B 16.8316,C -0.4652,E1 16.8954,E2 381.4109} C_DIS
LIN {X 48.241,Y 118.7992,Z 154,A 65.9012,B 16.8315,C -0.468,E1 16.8994,E2 382.9502} C_DIS
LIN {X 51.3488,Y 117.4899,Z 154,A 64.2876,B 16.8316,C -0.4628,E1 16.9035,E2 384.5761} C_DIS
LIN {X 54.8233,Y 115.9093,Z 154,A 62.733,B 16.8316,C -0.4659,E1 16.9074,E2 386.1138} C_DIS
LIN {X 57.6472,Y 114.5315,Z 154,A 61.3342,B 16.8316,C -0.4643,E1 16.9109,E2 387.5122} C_DIS
LIN {X 60.527,Y 113.0369,Z 154,A 59.7669,B 16.8318,C -0.4584,E1 16.9148,E2 389.0931} C_DIS
LIN {X 64.039,Y 111.085,Z 154,A 57.9768,B 16.8318,C -0.456,E1 16.9192,E2 390.8831} C_DIS
LIN {X 67.2696,Y 109.159,Z 154,A 56.3366,B 16.8318,C -0.4549,E1 16.9231,E2 392.5191} C_DIS
LIN {X 70.6959,Y 106.9718,Z 154,A 54.6134,B 16.8318,C -0.4553,E1 16.9271,E2 394.2323} C_DIS
LIN {X 73.2958,Y 105.2072,Z 154,A 53.219,B 16.8318,C -0.4533,E1 16.9303,E2 395.626} C_DIS
LIN {X 76.3816,Y 102.989,Z 154,A 51.3794,B 16.8321,C -0.4455,E1 16.9345,E2 397.4824} C_DIS
LIN {X 79.8703,Y 100.3073,Z 154,A 49.5169,B 16.8321,C -0.4456,E1 16.9386,E2 399.334} C_DIS
LIN {X 82.9039,Y 97.8151,Z 154,A 47.7092,B 16.8322,C -0.4405,E1 16.9425,E2 401.1486} C_DIS
LIN {X 86.104,Y 95.0101,Z 154,A 45.8769,B 16.8322,C -0.4392,E1 16.9463,E2 402.974} C_DIS
LIN {X 88.9833,Y 92.3194,Z 154,A 44.0395,B 16.8324,C -0.433,E1 16.95,E2 404.8211} C_DIS
LIN {X 92.3284,Y 88.9739,Z 154,A 41.9924,B 16.8324,C -0.4309,E1 16.954,E2 406.8618} C_DIS
LIN {X 95.0088,Y 86.1054,Z 154,A 40.2698,B 16.8325,C -0.4282,E1 16.9573,E2 408.582} C_DIS
LIN {X 97.601,Y 83.1557,Z 154,A 38.5164,B 16.8326,C -0.4244,E1 16.9605,E2 410.3365} C_DIS
LIN {X 100.1099,Y 80.1183,Z 154,A 36.7005,B 16.8328,C -0.4184,E1 16.9637,E2 412.16} C_DIS
LIN {X 102.6957,Y 76.7755,Z 154,A 34.8697,B 16.8328,C -0.416,E1 16.9668,E2 413.9856} C_DIS
LIN {X 104.8573,Y 73.7956,Z 154,A 33.3484,B 16.8328,C -0.4164,E1 16.9692,E2 415.494} C_DIS
LIN {X 106.9873,Y 70.6722,Z 154,A 31.5466,B 16.833,C -0.4082,E1 16.972,E2 417.3101} C_DIS
LIN {X 109.1066,Y 67.355,Z 154,A 29.8996,B 16.833,C -0.4078,E1 16.9745,E2 418.9459} C_DIS
LIN {X 111.1116,Y 63.993,Z 154,A 28.1434,B 16.8331,C -0.403,E1 16.977,E2 420.7045} C_DIS
LIN {X 112.7681,Y 61.0273,Z 154,A 26.6809,B 16.8331,C -0.401,E1 16.9789,E2 422.1619} C_DIS
LIN {X 114.2322,Y 58.2351,Z 154,A 25.2788,B 16.8333,C -0.3976,E1 16.9807,E2 423.5645} C_DIS
LIN {X 115.6394,Y 55.3883,Z 154,A 23.7717,B 16.8334,C -0.3906,E1 16.9826,E2 425.0832} C_DIS
LIN {X 117.2212,Y 51.9587,Z 154,A 22.2044,B 16.8334,C -0.3903,E1 16.9844,E2 426.6384} C_DIS
LIN {X 118.4316,Y 49.1362,Z 154,A 20.8349,B 16.8334,C -0.3866,E1 16.9859,E2 428.0089} C_DIS
LIN {X 119.629,Y 46.1449,Z 154,A 19.4174,B 16.8336,C -0.3834,E1 16.9873,E2 429.4253} C_DIS
LIN {X 120.7245,Y 43.1976,Z 154,A 18.0333,B 16.8336,C -0.3802,E1 16.9886,E2 430.8086} C_DIS
LIN {X 121.7483,Y 40.2217,Z 154,A 16.5209,B 16.8338,C -0.3723,E1 16.99,E2 432.3348} C_DIS
LIN {X 123.1476,Y 35.709,Z 154,A 14.4631,B 16.8339,C -0.3681,E1 16.9916,E2 434.3888} C_DIS
LIN {X 124.215,Y 31.7975,Z 154,A 12.7294,B 16.8339,C -0.3657,E1 16.9929,E2 436.1156} C_DIS
LIN {X 125.1115,Y 28.0667,Z 154,A 10.9022,B 16.8341,C -0.3565,E1 16.9941,E2 437.9578} C_DIS
LIN {X 125.9339,Y 24.1051,Z 154,A 9.2542,B 16.8341,C -0.357,E1 16.9949,E2 439.5896} C_DIS
LIN {X 126.4852,Y 21.0215,Z 154,A 7.869,B 16.8342,C -0.3533,E1 16.9956,E2 440.9747} C_DIS
LIN {X 127,Y 17.6537,Z 154,A 6.3747,B 16.8342,C -0.3498,E1 16.9962,E2 442.4677} C_DIS
LIN {X 127.3781,Y 14.6802,Z 154,A 5.0457,B 16.8344,C -0.3461,E1 16.9967,E2 443.7973} C_DIS
LIN {X 127.7493,Y 10.9809,Z 154,A 3.384,B 16.8344,C -0.341,E1 16.9971,E2 445.4611} C_DIS
LIN {X 127.9784,Y 7.8716,Z 154,A 1.9261,B 16.8346,C -0.3344,E1 16.9974,E2 446.9283} C_DIS
LIN {X 128.167,Y 3.7011,Z 154,A 0.2089,B 16.8346,C -0.3342,E1 16.9976,E2 448.6308} C_DIS
LIN {X 128.2223,Y 0.2724,Z 154,A -1.4417,B 16.8348,C -0.3251,E1 16.9976,E2 450.2971} C_DIS
LIN {X 128.1825,Y -3.1414,Z 154,A -2.952,B 16.8348,C -0.321,E1 16.9976,E2 451.8077} C_DIS
LIN {X 128.0281,Y -7.0439,Z 154,A -4.661,B 16.8349,C -0.317,E1 16.9973,E2 453.5149} C_DIS
LIN {X 127.7989,Y -10.3944,Z 154,A -6.0952,B 16.8349,C -0.3148,E1 16.997,E2 454.9434} C_DIS
LIN {X 127.438,Y -14.1483,Z 154,A -7.7474,B 16.835,C -0.3109,E1 16.9965,E2 456.5941} C_DIS
LIN {X 127.0549,Y -17.2579,Z 154,A -9.1324,B 16.835,C -0.3072,E1 16.996,E2 457.9793} C_DIS
LIN {X 126.5965,Y -20.3544,Z 154,A -10.5501,B 16.8352,C -0.3022,E1 16.9954,E2 459.4012} C_DIS
LIN {X 125.9314,Y -24.1179,Z 154,A -12.2602,B 16.8352,C -0.297,E1 16.9946,E2 461.1139} C_DIS
LIN {X 125.1042,Y -28.0988,Z 154,A -14.0271,B 16.8353,C -0.2933,E1 16.9935,E2 462.8776} C_DIS
LIN {X 124.3781,Y -31.1548,Z 154,A -15.4517,B 16.8354,C -0.2883,E1 16.9926,E2 464.3065} C_DIS
LIN {X 123.4009,Y -34.8235,Z 154,A -17.1227,B 16.8354,C -0.2841,E1 16.9914,E2 465.9769} C_DIS
LIN {X 122.2327,Y -38.725,Z 154,A -19.0578,B 16.8356,C -0.2745,E1 16.9898,E2 467.928} C_DIS
LIN {X 120.945,Y -42.5798,Z 154,A -20.8588,B 16.8357,C -0.2697,E1 16.9881,E2 469.7299} C_DIS
LIN {X 119.2878,Y -47.0226,Z 154,A -22.8009,B 16.8357,C -0.27,E1 16.9862,E2 471.6544} C_DIS
LIN {X 118.1031,Y -49.9229,Z 154,A -24.1894,B 16.8357,C -0.2664,E1 16.9847,E2 473.0436} C_DIS
LIN {X 116.6811,Y -53.1635,Z 154,A -25.8313,B 16.8359,C -0.2597,E1 16.9828,E2 474.6948} C_DIS
LIN {X 115.2335,Y -56.2305,Z 154,A -27.2479,B 16.8359,C -0.259,E1 16.9811,E2 476.102} C_DIS
LIN {X 113.9992,Y -58.6927,Z 154,A -28.532,B 16.8359,C -0.2536,E1 16.9795,E2 477.3941} C_DIS
LIN {X 112.3324,Y -61.8253,Z 154,A -30.0426,B 16.8359,C -0.2519,E1 16.9775,E2 478.8982} C_DIS
LIN {X 110.8338,Y -64.473,Z 154,A -31.5539,B 16.8361,C -0.2427,E1 16.9754,E2 480.429} C_DIS
LIN {X 108.6769,Y -68.046,Z 154,A -33.251,B 16.8361,C -0.2438,E1 16.9729,E2 482.1092} C_DIS
LIN {X 106.9772,Y -70.6876,Z 154,A -34.6412,B 16.8361,C -0.2405,E1 16.9708,E2 483.4997} C_DIS
LIN {X 105.2132,Y -73.2871,Z 154,A -36.0369,B 16.8361,C -0.2372,E1 16.9686,E2 484.8965} C_DIS
LIN {X 103.3688,Y -75.8663,Z 154,A -37.4335,B 16.8362,C -0.2343,E1 16.9663,E2 486.2926} C_DIS
LIN {X 101.0795,Y -78.8917,Z 154,A -39.2792,B 16.8364,C -0.2246,E1 16.9631,E2 488.1581} C_DIS
LIN {X 98.4064,Y -82.2013,Z 154,A -41.1074,B 16.8364,C -0.2225,E1 16.9599,E2 489.9804} C_DIS
LIN {X 95.7389,Y -85.2936,Z 154,A -42.8916,B 16.8364,C -0.2196,E1 16.9566,E2 491.7623} C_DIS
LIN {X 93.0854,Y -88.1816,Z 154,A -44.6173,B 16.8364,C -0.2164,E1 16.9533,E2 493.4872} C_DIS
LIN {X 90.4341,Y -90.8983,Z 154,A -46.3279,B 16.8365,C -0.212,E1 16.95,E2 495.2016} C_DIS
LIN {X 87.4959,Y -93.73,Z 154,A -48.1181,B 16.8365,C -0.2092,E1 16.9464,E2 496.9903} C_DIS
LIN {X 84.5867,Y -96.3641,Z 154,A -49.9333,B 16.8366,C -0.2032,E1 16.9425,E2 498.8149} C_DIS
LIN {X 81.3439,Y -99.1163,Z 154,A -51.7545,B 16.8366,C -0.202,E1 16.9387,E2 500.6291} C_DIS
LIN {X 78.2553,Y -101.573,Z 154,A -53.5973,B 16.8367,C -0.1957,E1 16.9346,E2 502.4833} C_DIS
LIN {X 75.1078,Y -103.9214,Z 154,A -55.1815,B 16.8367,C -0.1983,E1 16.9311,E2 504.0497} C_DIS
LIN {X 72.5384,Y -105.7308,Z 154,A -56.5745,B 16.8367,C -0.1961,E1 16.9279,E2 505.443} C_DIS
LIN {X 69.9255,Y -107.4768,Z 154,A -57.9687,B 16.8367,C -0.1939,E1 16.9246,E2 506.8377} C_DIS
LIN {X 67.2723,Y -109.1574,Z 154,A -59.3669,B 16.8367,C -0.1916,E1 16.9213,E2 508.2368} C_DIS
LIN {X 63.9922,Y -111.1121,Z 154,A -61.1328,B 16.8368,C -0.1866,E1 16.917,E2 510.0116} C_DIS
LIN {X 60.9709,Y -112.7984,Z 154,A -62.7451,B 16.8368,C -0.1818,E1 16.9131,E2 511.6332} C_DIS
LIN {X 57.1427,Y -114.7835,Z 154,A -64.6134,B 16.8368,C -0.1809,E1 16.9084,E2 513.4967} C_DIS
LIN {X 53.3929,Y -116.575,Z 154,A -66.3732,B 16.8368,C -0.1816,E1 16.904,E2 515.2471} C_DIS
LIN {X 50.526,Y -117.8457,Z 154,A -67.7694,B 16.8368,C -0.1798,E1 16.9004,E2 516.6439} C_DIS
LIN {X 47.6055,Y -119.0554,Z 154,A -69.1734,B 16.8368,C -0.1783,E1 16.8968,E2 518.0484} C_DIS
LIN {X 44.055,Y -120.4154,Z 154,A -70.9971,B 16.837,C -0.1719,E1 16.892,E2 519.8881} C_DIS
LIN {X 40.2022,Y -121.7548,Z 154,A -72.7952,B 16.837,C -0.1706,E1 16.8872,E2 521.685} C_DIS
LIN {X 36.3255,Y -122.9671,Z 154,A -74.6169,B 16.837,C -0.1685,E1 16.8823,E2 523.509} C_DIS
LIN {X 32.023,Y -124.1577,Z 154,A -76.5476,B 16.837,C -0.1688,E1 16.8772,E2 525.4339} C_DIS
Enddeposition()
END
